// TIA Portal project "N029_Testy Przekladni" (V17)

(* hardware
DEVICE "S7-1200 station_1"  S7-1200 Station
   slot 0: "Rack_0"  S7-1200 Rack  Rack  V1.0
   slot 1: "PLC"  CPU 1212C DC/DC/DC  6ES7 212-1AE40-0XB0  V4.5
DEVICE "HMI"  TP1200 Comfort
   slot 0: "HMI"  TP1200 Comfort  6AV2 124-0MC01-0AX0  17.0.0.0
   slot 1: "HMI_RT_1"  TP1200 Comfort  6AV2 124-0MC01-0AX0  17.0.0.0
   slot 5: "HMI.IE_CP_1"  PROFINET Interface  17.0.0.0
      slot 1: "PROFINET Interface_1"  PROFINET Interface
         slot 1: "Port_1"  Port
         slot 2: "Port_2"  Port
   slot 7: "HMI.MPI/DP_CP_1"  MPI/DP Interface  17.0.0.0
DEVICE "GSD device_1"  GSD.Device.PN
   slot 0: "Rack"  Rack  V1.0
   slot 0: "SK550P-PNT"  SK 550P-PNT
      slot 0: "SK 550P-PNT"  SK 550P-PNT
      slot 1: "PN-IO"  PN-IO
         slot 1: "Port 1 - RJ45 Connector 1"  Port 1 - RJ45 Connector 1
         slot 2: "Port 2 - RJ45 Connector 2"  Port 2 - RJ45 Connector 2
   slot 3: "PPO 4 (4 words)_1"  PPO 4 (4 words)
      slot 0: "PPO 4 (4 words)"  PPO 4 (4 words)
DEVICE "SCALANCE X005"  SCALANCE X-Station
   slot 0: "SCALANCE X rack"  Rail
   slot 0: "Switch_1"  6GK5 005-0BA00-1AB2  V1.0
*)

// ===== PLC "PLC"  CPU 1212C DC/DC/DC =====

VAR_GLOBAL   // PLC tag table "Default tag table"
   "Clock_Byte" AT %MB101 : Byte;
   "Clock_10Hz" AT %M101.0 : Bool;
   "Clock_5Hz" AT %M101.1 : Bool;
   "Clock_2.5Hz" AT %M101.2 : Bool;
   "Clock_2Hz" AT %M101.3 : Bool;
   "Clock_1.25Hz" AT %M101.4 : Bool;
   "Clock_1Hz" AT %M101.5 : Bool;
   "Clock_0.625Hz" AT %M101.6 : Bool;
   "Clock_0.5Hz" AT %M101.7 : Bool;
   "System_Byte" AT %MB100 : Byte;
   "FirstScan" AT %M100.0 : Bool;
   "DiagStatusUpdate" AT %M100.1 : Bool;
   "AlwaysTRUE" AT %M100.2 : Bool;
   "AlwaysFALSE" AT %M100.3 : Bool;
   "HMI_screen_no" AT %MB96 : USInt;
   "RUN_AUTO_mode" AT %M10.0 : Bool;
   "HMI_AUTO_Start_auto" AT %M10.2 : Bool;
   "HMI_Stop_auto" AT %M10.3 : Bool;
   "RUN_MANUAL_mode" AT %M10.1 : Bool;
   "MANUAL_direction" AT %M10.4 : Bool;
   "HMI_MANUAL_Start" AT %M10.5 : Bool;
END_VAR

VAR_GLOBAL   // PLC tag table "IOs_tags"
   "IN_pb_Reset" AT %I0.4 : Bool;
   "IN_pb_Start" AT %I0.0 : Bool;
   "OUT_green_LED" AT %M151.5 : Bool;
   "OUT_yellow_LED" AT %M151.6 : Bool;
   "OUT_red_LED" AT %M151.7 : Bool;
   "IN_pb_Gate_2_open" AT %I0.3 : Bool;
   "OUT_Gate_locks" AT %M151.0 : Bool;
   "OUT_pb_Reset_LED" AT %M151.1 : Bool;
   "OUT_pb_Start_LED" AT %M151.2 : Bool;
   "IN_pb_Stop" AT %I0.1 : Bool;
   "AIN_set_speed" AT %IW64 : Int;
   "IN_safety_lock_gate1" AT %I0.5 : Bool;
   "IN_safety_lock_gate2" AT %I0.6 : Bool;
   "IN_pb_Gate_1_open" AT %I0.2 : Bool;
END_VAR

// folder: Common

TYPE "typeDiagnostics"
TITLE = typeDiagnostics
// Provides a structure for detailed diagnostics
   STRUCT
      status : Word;   // Status of the block or error identification when error occurred
      subfunctionStatus : DWord;   // Status or return value of called FBs, FCs and system blocks
      stateNumber : DInt;   // State in the state machine of the block where the error occurred
   END_STRUCT;
END_TYPE

// folder: (top level)

DATA_BLOCK "Prozess_PPO2/4_DB"   // DB2
{ S7_Optimized_Access := 'TRUE' }
VERSION : 0.1
// stored: InstanceOfName Prozess_PPO2/4
"Prozess_PPO2/4"
BEGIN
END_DATA_BLOCK

DATA_BLOCK "Recipe_db"   // DB3
{ S7_Optimized_Access := 'TRUE' }
VERSION : 0.1
   VAR
      Velocity_array : Array[0..13] of Int;
      Time_array : Array[0..13] of Int;
      Set_speed : Int;
      Manual_speed : Int;
      Cumulated_time_array : Array[0..13] of Int;
   END_VAR
BEGIN
END_DATA_BLOCK

DATA_BLOCK "PLC_ variables"   // DB5
{ S7_Optimized_Access := 'TRUE' }
VERSION : 0.1
   VAR RETAIN
      RESET_state : USInt;
      STANDBY_state : USInt := 1;
      CHECK_LOCKS_state : USInt := 4;
      AUTO_state : USInt := 2;
      MANUAL_State : USInt := 3;
   END_VAR
   VAR
      STATE_machine_step : USInt;
      Measured_speed : Int;
   END_VAR
BEGIN
END_DATA_BLOCK

DATA_BLOCK "Auto_mode_DB"   // DB6
{ S7_Optimized_Access := 'TRUE' }
VERSION : 0.1
// stored: InstanceOfName Auto_mode
"Auto_mode"
BEGIN
END_DATA_BLOCK

// folder: System blocks/Program resources

DATA_BLOCK "IEC_Timer_0_DB"   // DB4
{ S7_Optimized_Access := 'TRUE' }
AUTHOR : Simatic
FAMILY : IEC
NAME : IEC_TMR
VERSION : 1.0
// stored: InstanceOfName IEC_TIMER
"IEC_TIMER"
BEGIN
END_DATA_BLOCK

DATA_BLOCK "time_from_Start_timer_DB"   // DB7
{ S7_Optimized_Access := 'TRUE' }
AUTHOR : Simatic
FAMILY : IEC
NAME : UDCNTR
VERSION : 1.2
// stored: InstanceOfName IEC_UDCOUNTER
"IEC_UDCOUNTER"
BEGIN
END_DATA_BLOCK

DATA_BLOCK "IEC_Counter_0_DB"   // DB8
{ S7_Optimized_Access := 'TRUE' }
AUTHOR : Simatic
FAMILY : IEC
NAME : CNTR
VERSION : 1.0
// stored: InstanceOfName IEC_COUNTER
"IEC_COUNTER"
BEGIN
END_DATA_BLOCK

DATA_BLOCK "IEC_Timer_0_DB_1"   // DB9
{ S7_Optimized_Access := 'TRUE' }
AUTHOR : Simatic
FAMILY : IEC
NAME : IEC_TMR
VERSION : 1.0
// stored: InstanceOfName IEC_TIMER
"IEC_TIMER"
BEGIN
END_DATA_BLOCK

// folder: (top level)

FUNCTION_BLOCK "Auto_mode"   // FB1, LAD
{ S7_Optimized_Access := 'TRUE' }
VERSION : 0.1
   VAR_OUTPUT
      Set_speed : Int;
   END_VAR
   VAR
      "60sec_marker" : Bool;
      STOPPED : USInt := 3;
      BRAKE : USInt := 2;
      RUN : USInt := 1;
      PREPARE_VAL : USInt;
      Time_from_start : UDInt;
      Time_for_next_step : UDInt;
      State : USInt;
   END_VAR
   VAR_TEMP
      "60sec" : Bool;
      timer_reset_marker : Bool;
      Time_curr_step : Int;
      Time_next_step : Int;
      i : Int;
      Curr_set_velocity : Int;
      Next_set_velocity : Int;
      j : Int;
      dVelocity : Int;
      Time_Step : Real;
      dTime : Real;
   END_VAR
BEGIN

REGION Network 1
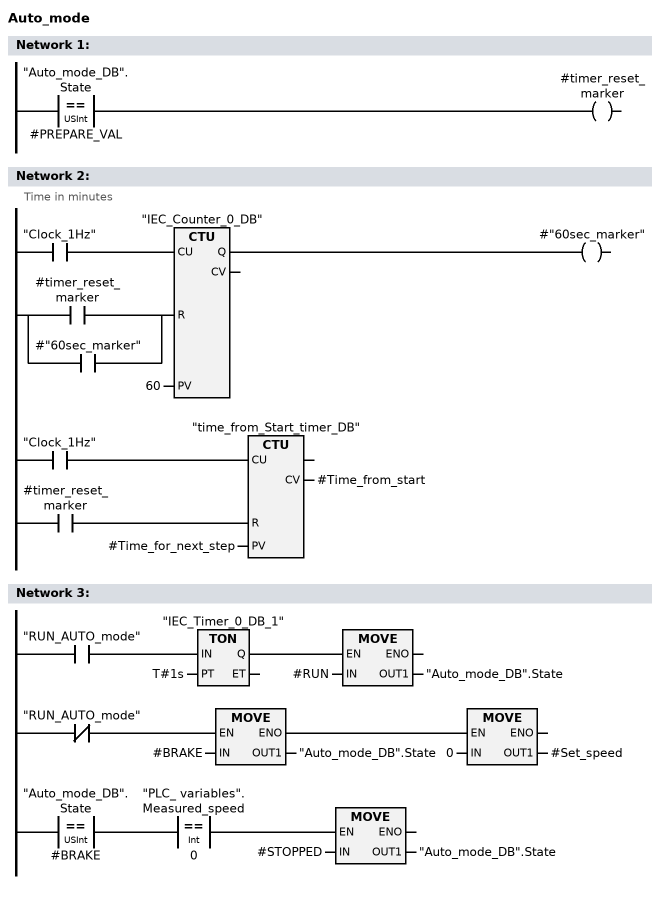
   RUNG wire#powerrail
      { S7_Templates := "SrcType := USInt" } EQ_Contact(in1 := "Auto_mode_DB".State, in2 := #PREPARE_VAL)
      Coil( #timer_reset_marker )
   END_RUNG
   // the same network as SCL:
   #timer_reset_marker := "Auto_mode_DB".State = #PREPARE_VAL;
END_REGION

REGION Network 2
   // Time in minutes
   "IEC_Counter_0_DB".CTU(CU := "Clock_1Hz", R := #timer_reset_marker OR #"60sec_marker", PV := 60);
   #"60sec_marker" := "IEC_Counter_0_DB".Q;
   "time_from_Start_timer_DB".CTU(CU := "Clock_1Hz",
                           R := #timer_reset_marker,
                           PV := #Time_for_next_step,
                           CV => #Time_from_start);
END_REGION

REGION Network 3
   "IEC_Timer_0_DB_1".TON(IN := "RUN_AUTO_mode", PT := T#1s);
   IF "IEC_Timer_0_DB_1".Q THEN "Auto_mode_DB".State := #RUN; END_IF;
   IF NOT "RUN_AUTO_mode" THEN
       "Auto_mode_DB".State := #BRAKE;
       #Set_speed := 0;
   END_IF;
   IF ("Auto_mode_DB".State = #BRAKE) AND ("PLC_ variables".Measured_speed = 0) THEN
       "Auto_mode_DB".State := #STOPPED;
   END_IF;
END_REGION

REGION Network 4 (SCL)
   IF (#State = #RUN OR #State = #PREPARE_VAL) THEN

       "Recipe_db".Cumulated_time_array[0] := 0;

       FOR #i := 0 TO 12 BY 1 DO
           "Recipe_db".Cumulated_time_array[#i + 1] := "Recipe_db".Cumulated_time_array[#i] + "Recipe_db".Time_array[#i + 1];
       END_FOR;

       FOR #j := 0 TO 12 BY 1 DO
           IF (#Time_from_start < ("Recipe_db".Cumulated_time_array[#j + 1] * 60)) THEN
               #Time_curr_step := "Recipe_db".Cumulated_time_array[#j] * 60;
               #Time_next_step := "Recipe_db".Cumulated_time_array[#j + 1] * 60;
               #Curr_set_velocity := "Recipe_db".Velocity_array[#j];
               #Next_set_velocity := "Recipe_db".Velocity_array[#j + 1];
               EXIT;
           ELSIF  (#Time_from_start > ("Recipe_db".Cumulated_time_array[#j + 1] * 60) AND #i=12) THEN
               #State:=#BRAKE;
           END_IF;
       END_FOR;

       #dTime := UDINT_TO_REAL(#Time_from_start - INT_TO_UDINT(#Time_curr_step));
       #Time_Step := (#Time_next_step - #Time_curr_step);
       #dVelocity := (#Next_set_velocity - #Curr_set_velocity);
       #Set_speed := #Curr_set_velocity + REAL_TO_INT(#dVelocity * (#dTime / #Time_Step));
   END_IF;
END_REGION
END_FUNCTION_BLOCK

FUNCTION_BLOCK "Prozess_PPO2/4"   // FB2, SCL
TITLE = PPO2/4
{ S7_Optimized_Access := 'TRUE' }
VERSION : 0.1
   VAR_INPUT
      HW_Identifier : Hw_Io;   // unique system constant created automatically by the system
      FI_Systembus : Int := 1;   // for frequency inverters in a system bus (1..8)
      Enable : Bool;   // 1 = enable drive
      Disable_Voltage : Bool;   // 1 = disable voltage
      Quick_Stop : Bool;   // 1 = quick stop
      Fault_ACK : Bool;   // 0 -> 1 fault acknowledgement
      Function_CTW_8 : Bool;   // bus controlword bit 8
      Function_CTW_9 : Bool;   // bus controlword bit 9
      Direction : Bool;   // 0 = cw / 1 = ccw
      Parameter_Set : Int;   // set of parameter (1..4)
      Setpoint_1 : Int;   // value setpoint 1
      Setpoint_2 : Int;   // value setpoint 2
      Setpoint_3 : Int;   // value setpoint 3
      Setpoint_32_Bit : Bool;   // 0 = setpoint 2 (16 bit) + setpoint 3 (16 bit) / 1 = setpoint 2 + 3 (32 bit)
      Setpoint_2_3 : DInt;   // value setpoint 2 + 3 (32 bit)
   END_VAR
   VAR_OUTPUT
      Not_Ready_to_Switch_On : Bool;   // inverter in not ready to switch-on state
      Switch_On_Inhibit : Bool;   // inverter in switch-on inhibit state
      Ready_to_Switch_On : Bool;   // inverter in ready to switch-on state
      Operation_Enabled : Bool;   // inverter in operation enabled state
      Fault : Bool;   // inverter in fault state
      Fault_Active : Bool;   // inverter in fault active state
      Quick_Stop_Active : Bool;   // inverter in quick stop active state
      Warning : Bool;   // warning identified
      Function_STW_10 : Bool;   // bus statusword bit 10
      Function_STW_13 : Bool;   // bus statusword bit 13
      Actual_Parameter_Set : Int;   // actual set of parameter 1..4
      Statusword : Word;   // statusword from inverter
      Actual_Value_1 : Int;   // actual value 1
      Actual_Value_2 : Int;   // actual value 2
      Actual_Value_3 : Int;   // actual value 3
      Actual_Value_2_3 : DInt;   // actual value 2 + 3 (32 bit)
   END_VAR
   VAR
      Controlword_Static : Word;   // controlword (to inverter)
      Control AT Controlword_Static : Struct   // definition controlword bits
         Start_Function_CTW_8 : Bool;   // set controlword bit 8
         Start_Function_CTW_9 : Bool;   // set controlword bit 9
         PZD_Valid : Bool;   // 0 = the transmitted data are invalid; 1 = the bus master transfers valid process data
         Rotatation_CW : Bool;   // 1 = switch on clockwise rotation
         Rotatation_CCW : Bool;   // 1 = switch on counter clockwise rotation
         Reserved : Bool;   // reserved
         Parameter_Set_Bit_0 : Bool;   // bit 0 of parameter set selection
         Parameter_Set_Bit_1 : Bool;   // bit 1 of parameter set selection
         Ready_for_Operation : Bool;   // 0 = reverse with break ramp, with voltage enabled at f=0Hz; 1 = set the frequency inverter to standby
         Disable_Voltage : Bool;   // 0 = switch off the output voltage; 1 = cancel "disable voltage"
         Quick_Stop : Bool;   // 0 = quick stop with programmed quick stop time; 1 = cancel "quick stop"
         Enable_Operation : Bool;   // 0 = block voltage; 1 = enable output voltage acceleration to acual setpoint
         Enable_Pulses : Bool;   // 0 = disable frequency inverter pulses; 1 = enable frequency inverter pulses
         Enable_Ramp : Bool;   // 0 = freeze actual frequency; 1 = enable frequency ramp
         Enable_Setpoint : Bool;   // 0 = set the setpoint to zero; 1 = use actual setpoint
         Acknowledge_the_Error : Bool;   // with the switch from 0 to 1, inactive errors are acknowledged
      END_STRUCT;
      GeoAddr : GEOADDR;   // geoaddr of the slot
      Get_GeoAddr : GEOADDR;   // geoaddr of the ~head module
      Statusword_Static : Word;   // statusword (from inverter)
      Status AT Statusword_Static : Struct   // definition statusword bits
         Setpoint_Reached : Bool;   // 0 = actual value does not correspond to the setpoint; 1 = actual value matches the setpoint
         Bus_Control : Bool;   // 0 = control on local device active; 1 = the master has been requested to take over control
         Function_STW_10 : Bool;   // function statusword bit 10 is active
         Rotatation_CW : Bool;   // 1 = the rotating field is clockwise
         Rotatation_CCW : Bool;   // 1 = the rotating field is counter-clockwise
         Function_STW_13 : Bool;   // function statusword bit 13 is active
         Parameter_Set_Bit_0 : Bool;   // bit 0 of the actual parameter set
         Parameter_Set_Bit_1 : Bool;   // bit 1 of the actual parameter set
         Ready_to_Switch_On : Bool;   // 1 = initialisation completed, charging relay switched on, output voltage disabled
         Ready : Bool;   // 0 = no switch-on command present or there is a fault; 1 = there is a switch-on command and there is no fault
         Operation_Enabled : Bool;   // 1 = the output voltage is enabled
         Fault : Bool;   // 0 = no fault 1 = the frequency inverter is in fault
         Voltage_Enabled : Bool;   // 0 = "disable voltage" command present
         Quick_Stop : Bool;   // 0 = "quick stop" command present
         Switch_On_Inhibit : Bool;   // 1 = with the command "shut down" the frequency inverter goes into state "ready to switch-on"
         Warning : Bool;   // 0 = no warning; 1 = active warning; drive operation continues, no acknowledgement necessary
      END_STRUCT;
   END_VAR
   VAR_TEMP
      Input_Address : DInt;   // input address of bus module
      Iw_Fi : UDInt;   // input start address from hardware configurator
      Iw_Fi_Length : UDInt;   // number of input bytes
      Laddr : Hw_Any;   // slot hw address
      Output_Address : DInt;   // output address of bus module
      Qw_Fi : UDInt;   // output start address from hardware configurator
      Qw_Fi_Length : UDInt;   // number of output bytes
      Ret_Geo2Log : Int;   // gro2log error information
      Ret_Log2Geo : Int;   // log2geo error information
      Ret_Rd_Addr : Int;   // rd_addr error information
   END_VAR
   VAR CONSTANT
      NOT_READY_TO_SWITCH_ON_MASK : Word := 2#1001111;   // status word mask for not ready to switch on
      NOT_READY_TO_SWITCH_ON_STATE : Word := 2#0000000;   // decoded fi status not ready to switch on
      SWITCH_ON_INHIBIT_MASK : Word := 2#1001111;   // status word mask for switch on inhibit
      SWITCH_ON_INHIBIT_STATE : Word := 2#1000000;   // decoded fi status switch on inhibit
      READY_TO_SWITCH_ON_MASK : Word := 2#1111111;   // status word mask for ready to swtich on
      READY_TO_SWITCH_ON_STATE : Word := 2#0110001;   // decoded fi status ready to swtich on
      SWITCHED_ON_MASK : Word := 2#1111111;   // status word mask for switched on
      SWITCHED_ON_STATE : Word := 2#0110011;   // decoded fi status switched on
      OPERATION_ENABLED_MASK : Word := 2#1111111;   // status word mask for operation enabled
      OPERATION_ENABLED_STATE : Word := 2#0110111;   // decoded fi status operation enabled
      FAULT_MASK : Word := 2#1001111;   // status word mask for fault
      FAULT_STATE : Word := 2#0001000;   // decoded fi status fault
      FAULT_ACTIVE_MASK : Word := 2#1001111;   // status word mask for fault activ
      FAULT_ACTIVE_STATE : Word := 2#0001111;   // decoded fi status fault activ
      PPO2_LENGTH : Word := 16;   // length of a ppo2 frame
      PPO2_4_LENGTH_TU3_PBR : Word := 12;   // length of a ppo2 and ppo4 pzd frame for a sk tu3-pbr
      PPO4_LENGTH : Word := 8;   // length of a ppo4 frame
      PROFIBUS : UInt := 2;   // profibus dp geoaddr area
      PROFINET : UInt := 1;   // profinet io geoaddr area
      QUICK_STOP_ACTIVE_MASK : Word := 2#1111111;   // status word mask for quick stop activ
      QUICK_STOP_ACTIVE_STATE : Word := 2#0010111;   // decoded fi status quick stop activ
      SLOT_OFFSET_PBR : UInt := 1;   // profibus dp slot offset of bus module
      SLOT_OFFSET_PNT : UInt := 2;   // profinet io slot offset of bus module
   END_VAR
   // GeoAddr.HWTYPE := 4;
BEGIN
   // get area, io station and station from ~head module (hw address)
   #Ret_Log2Geo := LOG2GEO(LADDR := #HW_Identifier, GEOADDR := #Get_GeoAddr);
   #GeoAddr.AREA := #Get_GeoAddr.AREA;
   #GeoAddr.IOSYSTEM := #Get_GeoAddr.IOSYSTEM;
   #GeoAddr.STATION := #Get_GeoAddr.STATION;

   IF #Get_GeoAddr.AREA = #PROFINET THEN     // for profinet io
       #GeoAddr.SLOT := INT_TO_UINT(#FI_Systembus) + #SLOT_OFFSET_PNT;
   ELSIF #Get_GeoAddr.AREA = #PROFIBUS THEN  // for profibus dp
       #GeoAddr.SLOT := INT_TO_UINT(#FI_Systembus) + #SLOT_OFFSET_PBR;
   ELSE  // wrong area
       #Actual_Value_1 := 0;
       #Actual_Value_2 := 0;
       #Actual_Value_3 := 0;
       #Actual_Value_2_3 := 0;
       #Not_Ready_to_Switch_On := FALSE;
       #Switch_On_Inhibit := FALSE;
       #Ready_to_Switch_On := FALSE;
       #Operation_Enabled := FALSE;
       #Fault_Active := FALSE;
       #Fault := FALSE;
       #Quick_Stop_Active := FALSE;
       #Warning := FALSE;
       #Function_STW_10 := FALSE;
       #Function_STW_13 := FALSE;
       #Statusword := 0;
       #Actual_Parameter_Set := 0;
       RETURN;
   END_IF;

   // get slot hw address (systembus fi)
   #Ret_Geo2Log := GEO2LOG(GEOADDR := #GeoAddr, LADDR => #Laddr);
   // based on slot hw address get io addresses
   #Ret_Rd_Addr := RD_ADDR(LADDR := #Laddr, PIADDR => #Iw_Fi, PICount => #Iw_Fi_Length,
                           PQADDR => #Qw_Fi, PQCount => #Qw_Fi_Length);

   IF #Iw_Fi_Length = #PPO4_LENGTH THEN    // if PPO4 -> no PKW channel
       #Input_Address  := UDINT_TO_DINT(#Iw_Fi);
       #Output_Address := UDINT_TO_DINT(#Qw_Fi);
   ELSIF #Iw_Fi_Length = #PPO2_4_LENGTH_TU3_PBR AND
         #Get_GeoAddr.AREA = #PROFIBUS THEN // special case SK xU3-PBR: PPO2/4 -> 6 words/no PKW channel
       #Input_Address := UDINT_TO_DINT(#Iw_Fi);
       #Output_Address := UDINT_TO_DINT(#Qw_Fi);
   ELSIF #Iw_Fi_Length = #PPO2_LENGTH THEN  // else if PPO2 -> with PKW channel
       #Input_Address  := UDINT_TO_DINT(#Iw_Fi) + 8;
       #Output_Address := UDINT_TO_DINT(#Qw_Fi) + 8;
   ELSE // wrong PPO Type
       #Actual_Value_1 := 0;
       #Actual_Value_2 := 0;
       #Actual_Value_3 := 0;
       #Actual_Value_2_3 := 0;
       #Not_Ready_to_Switch_On := FALSE;
       #Switch_On_Inhibit := FALSE;
       #Ready_to_Switch_On := FALSE;
       #Operation_Enabled := FALSE;
       #Fault_Active := FALSE;
       #Fault := FALSE;
       #Quick_Stop_Active := FALSE;
       #Warning := FALSE;
       #Function_STW_10 := FALSE;
       #Function_STW_13 := FALSE;
       #Statusword := 0;
       #Actual_Parameter_Set := 0;
       RETURN;
   END_IF;

   // prepare controlword to inverter********************
   #Control.Ready_for_Operation    := #Enable;
   #Control.Disable_Voltage        := NOT #Disable_Voltage;
   #Control.Quick_Stop             := NOT #Quick_Stop;
   #Control.Enable_Operation       := TRUE;
   #Control.Enable_Pulses          := TRUE;
   #Control.Enable_Ramp            := TRUE;
   #Control.Enable_Setpoint        := TRUE;
   #Control.Acknowledge_the_Error  := #Fault_ACK;
   #Control.Start_Function_CTW_8   := #Function_CTW_8;
   #Control.Start_Function_CTW_9   := #Function_CTW_9;
   #Control.PZD_Valid              := TRUE;
   #Control.Rotatation_CCW         := #Direction;

   CASE #Parameter_Set OF
       1:  // statement section parameter set 1
           #Control.Parameter_Set_Bit_0 := FALSE;
           #Control.Parameter_Set_Bit_1 := FALSE;
       2:  // statement section parameter set 2
           #Control.Parameter_Set_Bit_0 := TRUE;
           #Control.Parameter_Set_Bit_1 := FALSE;
       3:  // statement section parameter set 3
           #Control.Parameter_Set_Bit_0 := FALSE;
           #Control.Parameter_Set_Bit_1 := TRUE;
       4:  // statement section parameter set 4
           #Control.Parameter_Set_Bit_0 := TRUE;
           #Control.Parameter_Set_Bit_1 := TRUE;
       ELSE  // default statement section parameter set 1
           #Control.Parameter_Set_Bit_0 := FALSE;
           #Control.Parameter_Set_Bit_1 := FALSE;
   END_CASE;

   // write controlword**********************************
   POKE(area := 16#82,
        dbNumber := 0,
        byteOffset := #Output_Address,
        value := #Controlword_Static);
   // write setpoints************************************
   POKE(area := 16#82,
        dbNumber := 0,
        byteOffset := #Output_Address + 2,
        value := INT_TO_WORD(#Setpoint_1));
   IF #Setpoint_32_Bit THEN
       POKE(area := 16#82,
            dbNumber := 0,
            byteOffset := #Output_Address + 4,
            value := DINT_TO_DWORD(#Setpoint_2_3));
   ELSE
       POKE(area := 16#82,
            dbNumber := 0,
            byteOffset := #Output_Address + 4,
            value := INT_TO_WORD(#Setpoint_2));
       POKE(area := 16#82,
            dbNumber := 0,
            byteOffset := #Output_Address + 6,
            value := INT_TO_WORD(#Setpoint_3));
   END_IF;

   // read statusword************************************
   #Statusword_Static := PEEK_WORD(area := 16#81, dbNumber := 0, byteOffset := #Input_Address);
   // read actual values*********************************
   #Actual_Value_1   := WORD_TO_INT(PEEK_WORD(area := 16#81, dbNumber := 0, byteOffset := #Input_Address + 2));
   #Actual_Value_2   := WORD_TO_INT(PEEK_WORD(area := 16#81, dbNumber := 0, byteOffset := #Input_Address + 4));
   #Actual_Value_3   := WORD_TO_INT(PEEK_WORD(area := 16#81, dbNumber := 0, byteOffset := #Input_Address + 6));
   #Actual_Value_2_3 := DWORD_TO_DINT(PEEK_DWORD(area := 16#81, dbNumber := 0, byteOffset := #Input_Address + 4));

   // decode statusword and set outputs******************
   #Not_Ready_to_Switch_On := (#Statusword_Static AND #NOT_READY_TO_SWITCH_ON_MASK) = #NOT_READY_TO_SWITCH_ON_STATE;
   #Switch_On_Inhibit      := (#Statusword_Static AND #SWITCH_ON_INHIBIT_MASK) = #SWITCH_ON_INHIBIT_STATE;
   #Ready_to_Switch_On     := (#Statusword_Static AND #READY_TO_SWITCH_ON_MASK) = #READY_TO_SWITCH_ON_STATE;
   #Operation_Enabled      := (#Statusword_Static AND #OPERATION_ENABLED_MASK) = #OPERATION_ENABLED_STATE;
   #Fault_Active           := (#Statusword_Static AND #FAULT_ACTIVE_MASK) = #FAULT_ACTIVE_STATE;
   #Fault                  := (#Statusword_Static AND #FAULT_MASK) = #FAULT_STATE;
   #Quick_Stop_Active      := (#Statusword_Static AND #QUICK_STOP_ACTIVE_MASK) = #QUICK_STOP_ACTIVE_STATE;
   #Warning                := #Status.Warning;
   #Function_STW_10        := #Status.Function_STW_10;
   #Function_STW_13        := #Status.Function_STW_13;
   #Statusword             := #Statusword_Static;
   #Actual_Parameter_Set   := WORD_TO_INT(SHR(IN := #Statusword_Static, N := 14)) + 1;
END_FUNCTION_BLOCK

FUNCTION "Manual_mode" : Void   // FC1, LAD
{ S7_Optimized_Access := 'TRUE' }
VERSION : 0.1
   VAR_OUTPUT
      Set_speed : Int;
   END_VAR
   VAR_TEMP
      calculated_speed : Real;
   END_VAR
   VAR CONSTANT
      MULTIPLY : Real := 0.2;
   END_VAR
BEGIN

REGION Network 1 (SCL)
   #calculated_speed := INT_TO_REAL("AIN_set_speed") * #MULTIPLY;
   #Set_speed := REAL_TO_INT(LIMIT_REAL(IN:=#calculated_speed,MN:= 0.0,MX:= 6000.0));
END_REGION
END_FUNCTION

ORGANIZATION_BLOCK "Main"   // OB1, LAD, ProgramCycle
TITLE = "Main Program Sweep (Cycle)"
{ S7_Optimized_Access := 'TRUE' }
VERSION : 0.1
   VAR_INPUT
      Initial_Call : Bool;   // Initial call of this OB
      Remanence : Bool;   // =True, if remanent data are available
   END_VAR
   VAR_TEMP   // added for the SCL form of the ladder/FBD networks
      _w1 : Bool;
   END_VAR
BEGIN

REGION Network 1: initial state
   // State machine
   // 1- reset state
   // 2- standby
   // 3- manual mode
   // 4- auto mode
   // 5- error
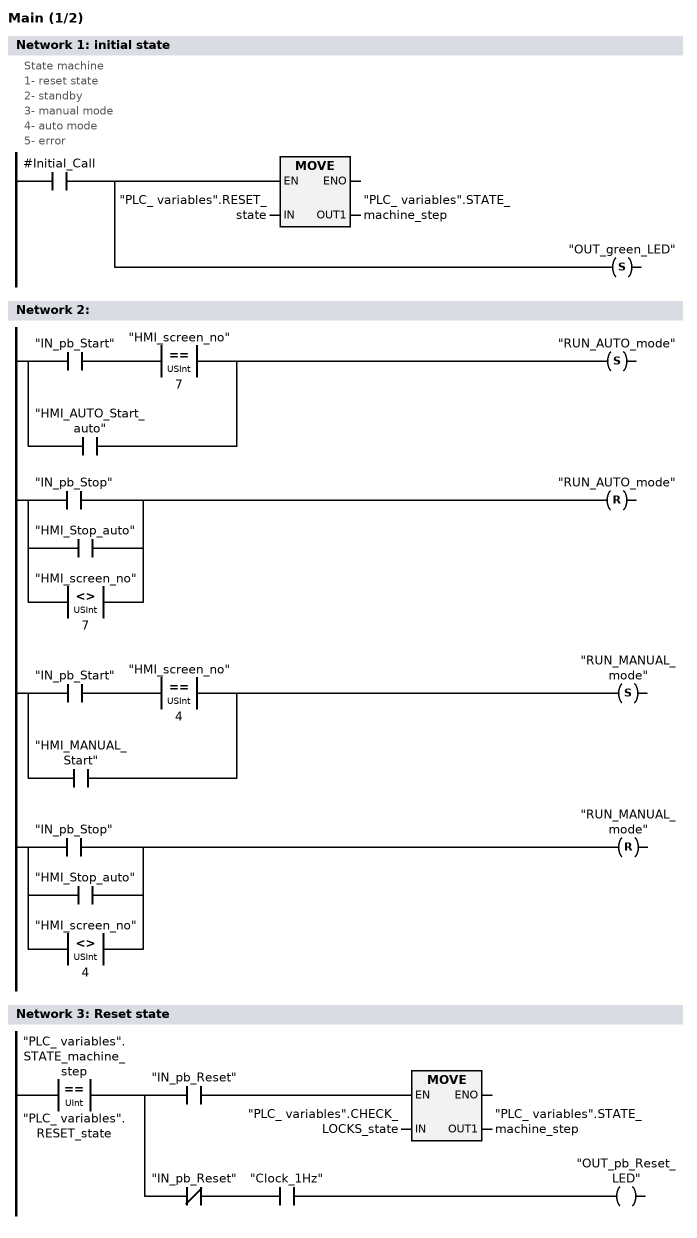
   RUNG wire#powerrail
      Contact( #Initial_Call )
      wire#w1
      Move(in := "PLC_ variables".RESET_state, out1 => "PLC_ variables".STATE_machine_step)
   END_RUNG
   RUNG wire#w1
      S_Coil( "OUT_green_LED" )
   END_RUNG
   // the same network as SCL:
   IF #Initial_Call THEN
       "PLC_ variables".STATE_machine_step := "PLC_ variables".RESET_state;
       "OUT_green_LED" := TRUE;
   END_IF;
END_REGION

REGION Network 2
   RUNG wire#powerrail
      Contact( "IN_pb_Start" )
      { S7_Templates := "SrcType := USInt" } EQ_Contact(in1 := "HMI_screen_no", in2 := 7)
      wire#w1
      S_Coil( "RUN_AUTO_mode" )
   END_RUNG
   RUNG wire#powerrail
      Contact( "HMI_AUTO_Start_auto" )
   END_RUNG wire#w1
   RUNG wire#powerrail
      Contact( "IN_pb_Stop" )
      wire#w2
      R_Coil( "RUN_AUTO_mode" )
   END_RUNG
   RUNG wire#powerrail
      Contact( "HMI_Stop_auto" )
   END_RUNG wire#w2
   RUNG wire#powerrail
      { S7_Templates := "SrcType := USInt" } NE_Contact(in1 := "HMI_screen_no", in2 := 7)
   END_RUNG wire#w2
   RUNG wire#powerrail
      Contact( "IN_pb_Start" )
      { S7_Templates := "SrcType := USInt" } EQ_Contact(in1 := "HMI_screen_no", in2 := 4)
      wire#w3
      S_Coil( "RUN_MANUAL_mode" )
   END_RUNG
   RUNG wire#powerrail
      Contact( "HMI_MANUAL_Start" )
   END_RUNG wire#w3
   RUNG wire#powerrail
      Contact( "IN_pb_Stop" )
      wire#w4
      R_Coil( "RUN_MANUAL_mode" )
   END_RUNG
   RUNG wire#powerrail
      Contact( "HMI_Stop_auto" )
   END_RUNG wire#w4
   RUNG wire#powerrail
      { S7_Templates := "SrcType := USInt" } NE_Contact(in1 := "HMI_screen_no", in2 := 4)
   END_RUNG wire#w4
   // the same network as SCL:
   IF ("IN_pb_Start" AND ("HMI_screen_no" = 7)) OR "HMI_AUTO_Start_auto" THEN
       "RUN_AUTO_mode" := TRUE;
   END_IF;
   IF "IN_pb_Stop" OR "HMI_Stop_auto" OR ("HMI_screen_no" <> 7) THEN "RUN_AUTO_mode" := FALSE; END_IF;
   IF ("IN_pb_Start" AND ("HMI_screen_no" = 4)) OR "HMI_MANUAL_Start" THEN "RUN_MANUAL_mode" := TRUE; END_IF;
   IF "IN_pb_Stop" OR "HMI_Stop_auto" OR ("HMI_screen_no" <> 4) THEN "RUN_MANUAL_mode" := FALSE; END_IF;
END_REGION

REGION Network 3: Reset state
   RUNG wire#powerrail
      { S7_Templates := "SrcType := UInt" } EQ_Contact(in1 := "PLC_ variables".STATE_machine_step, in2 := "PLC_ variables".RESET_state)
      wire#w1
      Contact( "IN_pb_Reset" )
      Move(in := "PLC_ variables".CHECK_LOCKS_state, out1 => "PLC_ variables".STATE_machine_step)
   END_RUNG
   RUNG wire#w1
      I_Contact( "IN_pb_Reset" )
      Contact( "Clock_1Hz" )
      Coil( "OUT_pb_Reset_LED" )
   END_RUNG
   // the same network as SCL:
   #_w1 := "PLC_ variables".STATE_machine_step = "PLC_ variables".RESET_state;
   IF #_w1 AND "IN_pb_Reset" THEN
       "PLC_ variables".STATE_machine_step := "PLC_ variables".CHECK_LOCKS_state;
   END_IF;
   "OUT_pb_Reset_LED" := #_w1 AND NOT "IN_pb_Reset" AND "Clock_1Hz";
END_REGION

REGION Network 5: Standby state
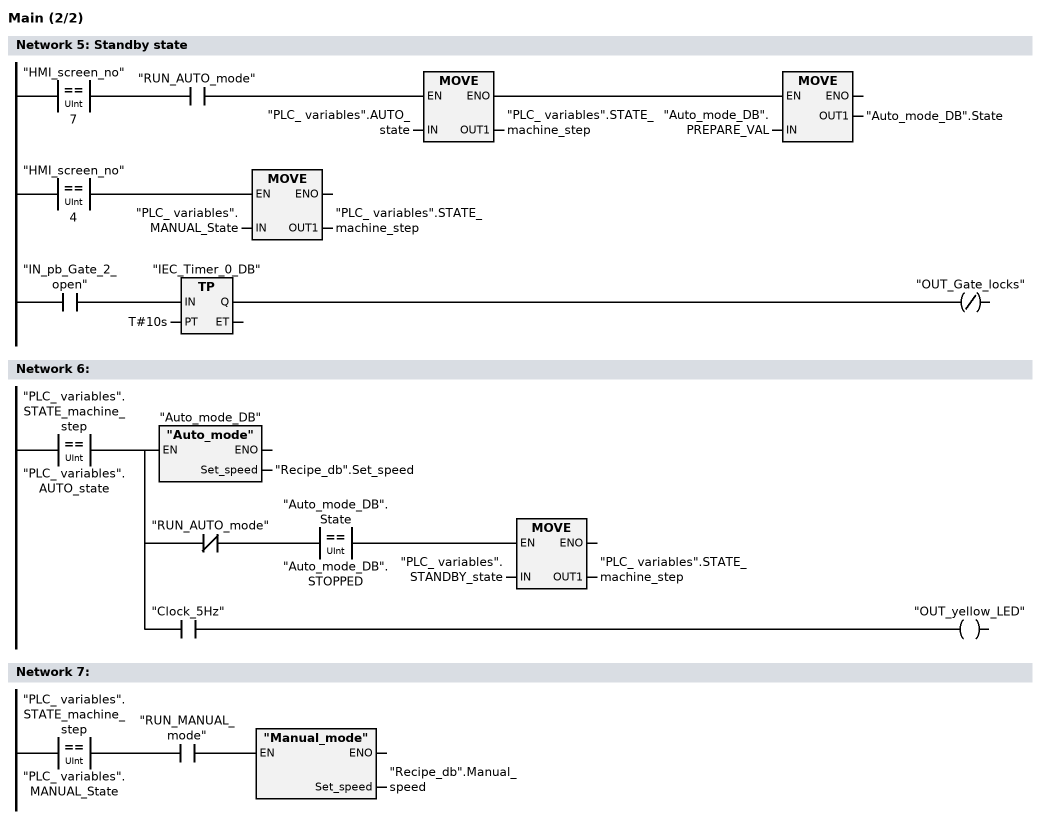
   IF ("HMI_screen_no" = 7) AND "RUN_AUTO_mode" THEN
       "PLC_ variables".STATE_machine_step := "PLC_ variables".AUTO_state;
       "Auto_mode_DB".State := "Auto_mode_DB".PREPARE_VAL;
   END_IF;
   IF "HMI_screen_no" = 4 THEN "PLC_ variables".STATE_machine_step := "PLC_ variables".MANUAL_State; END_IF;
   "IEC_Timer_0_DB".TP(IN := "IN_pb_Gate_2_open", PT := T#10s);
   "OUT_Gate_locks" := NOT "IEC_Timer_0_DB".Q;
END_REGION

REGION Network 6
   RUNG wire#powerrail
      { S7_Templates := "SrcType := UInt" } EQ_Contact(in1 := "PLC_ variables".STATE_machine_step, in2 := "PLC_ variables".AUTO_state)
      wire#w1
      "Auto_mode_DB"(Set_speed => "Recipe_db".Set_speed)
   END_RUNG
   RUNG wire#w1
      I_Contact( "RUN_AUTO_mode" )
      { S7_Templates := "SrcType := UInt" } EQ_Contact(in1 := "Auto_mode_DB".State, in2 := "Auto_mode_DB".STOPPED)
      Move(in := "PLC_ variables".STANDBY_state, out1 => "PLC_ variables".STATE_machine_step)
   END_RUNG
   RUNG wire#w1
      Contact( "Clock_5Hz" )
      Coil( "OUT_yellow_LED" )
   END_RUNG
   // the same network as SCL:
   #_w1 := "PLC_ variables".STATE_machine_step = "PLC_ variables".AUTO_state;
   IF #_w1 THEN
       "Auto_mode_DB"(Set_speed => "Recipe_db".Set_speed);   // "Auto_mode"
   END_IF;
   IF #_w1 AND NOT "RUN_AUTO_mode" AND ("Auto_mode_DB".State = "Auto_mode_DB".STOPPED) THEN
       "PLC_ variables".STATE_machine_step := "PLC_ variables".STANDBY_state;
   END_IF;
   "OUT_yellow_LED" := #_w1 AND "Clock_5Hz";
END_REGION

REGION Network 7
   RUNG wire#powerrail
      { S7_Templates := "SrcType := UInt" } EQ_Contact(in1 := "PLC_ variables".STATE_machine_step, in2 := "PLC_ variables".MANUAL_State)
      Contact( "RUN_MANUAL_mode" )
      "Manual_mode"(Set_speed => "Recipe_db".Manual_speed)
   END_RUNG
   // the same network as SCL:
   IF ("PLC_ variables".STATE_machine_step = "PLC_ variables".MANUAL_State) AND "RUN_MANUAL_mode" THEN
       "Manual_mode"(Set_speed => "Recipe_db".Manual_speed);
   END_IF;
END_REGION
END_ORGANIZATION_BLOCK

// ===== library types =====

// folder: LFTP

TYPE "LFTP_typeFtpParam"
TITLE = LFTP_typeFtpParam / LFTP_typeUserParam
VERSION : 0.1
// Data type for user parameters of the LFTP FB / Data type for user parameters of the LFTP_Client FB
   STRUCT
      ftpActiveMode : Bool;   // False: FTP mode is set to passive; True: FTP mode is set to active
      portActiveMode : UInt := 2001;   // Must be set >2000; Port for FTP-active mode data connection / Must be set >2000; Local Port for FTP active mode
      ftpCmd : Int;   // 2 STORE, 3 RETRIEVE, 4 DELETE, 6 APPEND
      filename : String;   // FTP Filename
   END_STRUCT;
END_TYPE

TYPE "LFTP_typeConnParam"
TITLE = LFTP_typeConnParam
// Datatype for the Parameters needed for connection to FTP-Server / Data type for connection parameters needed to establish a connection to the FTP server
   STRUCT
      hwID : HW_ANY;   // HW-identifier of IE-interface submodule
      serverAddress : String;   // Remote-Adress of FTP-Server / IP address or host name of FTP server
      username : String := '';   // Username of the FTP-Client / User name of the FTP client
      password : String := '';   // Password of the FTP-Client / Password of the FTP client
   END_STRUCT;
END_TYPE

FUNCTION_BLOCK "LFTP_Client"   // FB2, SCL
TITLE = LFTP_Client
{ S7_Optimized_Access := 'TRUE' }
AUTHOR : Siemens Industry Online Support
FAMILY : LFTP
VERSION : 6.0
// Implements an FTP client
   VAR_INPUT
      enable : Bool := FALSE;   // Enable client and connect to FTP server
      execute : Bool := FALSE;   // Execute FTP command
      timeOut : Time := T#5s;   // Time for watchdog
   END_VAR
   VAR_OUTPUT
      valid : Bool := FALSE;   // TRUE: Valid set of output values available at the FB
      done : Bool := FALSE;   // TRUE: Last command was successful
      busy : Bool := FALSE;   // TRUE: FB is not finished and new output values can be expected
      error : Bool := FALSE;   // TRUE: An error occurred during the execution of the FB
      status : Word := 16#7000;   // 16#0000 - 16#7FFF: Status of the FB, 16#8000 - 16#FFFF: Error identification
      diagnostics : "typeDiagnostics";   // Diagnostics information of FB
   END_VAR
   VAR_IN_OUT
      connParam : "LFTP_typeConnParam";   // Connection parameters
      ftpParam : "LFTP_typeFtpParam";   // FTP parameters
      dataLen : UDInt;   // Length of data to be sent or received
      data : Array[*] of Byte;   // Data to be sent or received
   END_VAR
   VAR
      statEnableOld : Bool;   // Last cycle's value of 'enable' input for edge detection
      statExecuteOld : Bool;   // Last cycle's value of 'execute' input for edge detection
      statValid : Bool;   // Static value for output 'valid'
      statDone : Bool;   // Static value for output 'done'
      statBusy : Bool;   // Static value for output 'busy'
      statError : Bool;   // Static value for output 'error'
      statErrorUserCleared : Bool;   // Error occurred that can only be solved by user; rising edge at enable input necessary
      statErrorAutoCleared : Bool;   // Error occurred that can be acknowledged by FB
      statStatus : Word := 16#7000;   // Static value for output 'status'
      statSubfunctionStatus : DWord;   // Status or return value of called FBs, FCs and system blocks
      statFBErrorState : DInt;   // State in the state machine of the block where the error occurred
      statFBState : UInt := 0;   // State in the state machine of the FB
      statDisablingCompleted : Bool;   // TRUE: Disabling has been completed
      statEmptyDiagnostics : "typeDiagnostics";   // Empty diagnostics information (for initialization purposes only)
      statConnParam : Struct   // Connection parameters
         isQDN : Bool;   // Is set to TRUE when connParam.url recognised as QDN
         paramControlQDN : TCON_QDN;   // Connection parameters in form of QDN
         paramControlIP : TCON_IP_v4;   // Connection parameters in form of IP address
         paramDataQDN : TCON_QDN;   // Connection parameters of data connection in form of QDN
         paramDataIP : TCON_IP_v4;   // Connection parameters of data connection in form of IP address
      END_STRUCT;
      statFtpParam : "LFTP_typeFtpParam";
      instTconSettingsControl : TCONSettings;
      statTconSettingsControlReq : Bool;
      statTconSettingsControlOption : TCON_TCPTermination;   // Set TCP Termination for control connection to "Graceful shutdown"
      instTconControl : TCON;   // Tcon for FTP control connection
      statTconControlReq : Bool := FALSE;
      instTsendControl : TSEND;   // Tsend for FTP control commands
      statTsendControlReq : Bool := FALSE;
      statTsendControlLen : UInt;   // Length of data to be sent over control connection
      instTrcvControl : TRCV;   // Trcv for receiving reply codes from FTP-Server
      statTrcvControlEnable : Bool;   // Enable TRCV for control connection
      instTdisconControl : TDISCON;   // TDiscon for control connection
      statTdisconControlReq : Bool := FALSE;
      instTconSettingsData : TCONSettings;
      statTconSettingsDataReq : Bool;
      statTconSettingsDataOption : TCON_TCPTermination;   // Set TCP Termination for data connection to "Graceful shutdown"
      instTconData : TCON;   // Tcon for FTP data connection
      statTconDataReq : Bool := FALSE;
      instTsendData : TSEND;   // Tsend for sending data to FTP-Server
      statTsendDataReq : Bool := FALSE;
      instTrcvData : TRCV;   // Trcv for receiving data from the FTP-Server
      statTrcvDataEnable : Bool;   // Enable TRCV for data connection
      instTdisconData : TDISCON;   // TDiscon for data connection
      statTdisconDataReq : Bool := FALSE;
      statCtrlReplyCode : Int;   // Reply code received from FTP-Server
      statTsendControlData : Array[0..100] of Char;   // Data for Tsend of control connection
      statTrcvControlData : Array[0..149] of Char;   // Data for Trcv of data connection
      statTrcvControlString : String;
      statLocalHighPort : UInt;   // Local port (LowPort*256 + HighPort)
      statLocalLowPort : UInt;   // Local port (LowPort*256 + HighPort)
      statIpAsString : String;   // Client IP-Adress as a String
      statLocalPortAsString : String;   // Local Port combined as String
      statPortPosition : Int;
      statSearchPosition : Int;
      statRemotePortLowStr : String;   // Remote LowPort for passive mode as String (LowPort*256 + HighPort)
      statRemotePortHighStr : String;   // Remote HighPort for passive mode as String (LowPort*256 + HighPort)
      statRemotePort : UInt;   // Combined remote port for passive mode
      statRcvDataBuffer : Array[0..8191] of Byte;
      statDataLen : UDInt;
      statCtrlConnectionID : Word;   // Connection ID of the control connection
      statDataConnectionID : Word;   // Connection ID of the data connection
      statCtrlConnEstablished : Bool;
      statDataConnEstablished : Bool;
      statUserCredentials : Struct
         username : String;
         password : String;
      END_STRUCT;
      instTimeout : TON_TIME;
      statTimeoutIn : Bool;
      instRdRec : RDREC;
      statRdRecRecord : Struct
         blockType : UInt;
         blockLength : UInt;
         blockVersionHigh : USInt;
         blockVersionLow : USInt;
         data : Array[0..#REC_IP_MLEN] of Byte;
      END_STRUCT;
   END_VAR
   VAR_TEMP
      tempUrl : String;
      tempPos : Int;
      tempString : String;
      tempIndex : DInt;
      tempRet : Word;   // Return value
      tempStartIpAddress : USInt;   // Start of IP address in data record
   END_VAR
   VAR CONSTANT
      FB_STATE_NO_PROCESSING : UInt := 0;   // FB state: No processing
      FB_STATE_EVAL_CONN_PARAM : UInt := 10;   // FB state: Evaluate connection parameters
      FB_STATE_GET_ID_CTRL : UInt := 11;   // FB state: Get connection ID for control connection
      FB_STATE_EST_CTRL_CONN : UInt := 20;   // FB state: Establish control connection
      FB_STATE_SEND_USERNAME : UInt := 30;   // FB state: Send FTP username
      FB_STATE_USERNAME_SENT : UInt := 31;   // FB state: FTP username sent, wait for reply code 331
      FB_STATE_SEND_PASSWORD : UInt := 32;   // FB state: Send password
      FB_STATE_PASSWORD_SENT : UInt := 33;   // FB state: Password sent, wait for reply code 230
      FB_STATE_SET_CON_TYPE : UInt := 34;   // FB state: Set type of FTP connection ("Type I")
      FB_STATE_TYPE_SENT : UInt := 35;   // FB state: Type of FTP connection SENT
      FB_STATE_CTRL_CONN_EST : UInt := 50;   // FB state: Control connection established
      FB_STATE_GET_ID_DATA : UInt := 51;   // FB state: Get connection ID for data connection
      FB_STATE_GET_IP_INFO : UInt := 52;   // FB state: Get IP of PLC for FTP active mode
      FB_STATE_SEND_FTP_MODE : UInt := 53;   // FB state: Send FTP mode
      FB_STATE_EST_DATA_CONN : UInt := 54;   // FB state: FTP mode sent, establishing data connection
      FB_STATE_SEND_FILENAME_CMD : UInt := 55;   // FB state: Send filename and FTP-command
      FB_STATE_FILENAME_CMD_SENT : UInt := 56;   // FB state: Filename and command sent
      FB_STATE_DATA_TRANSFER : UInt := 60;   // FB state: Data transfer
      FB_STATE_CLOSE_DATA_CON : UInt := 70;   // FB state: Close data connection
      FB_STATE_SEND_QUIT : UInt := 90;   // FB state: Send 'Quit' command
      FB_STATE_DISCONNECT_CTRL : UInt := 91;   // FB state: Close control connection
      STATUS_EXECUTION_FINISHED : Word := 16#0000;   // Execution finished without errors
      STATUS_NO_CALL : Word := 16#7000;   // FB in idle, no active connection
      STATUS_FIRST_CALL : Word := 16#7001;   // First call after incoming new job (rising edge 'enable')
      STATUS_ESTABLISH_CTRL_CON : Word := 16#7002;   // Establish control connection
      STATUS_DISCON_CONTRL_CON : Word := 16#7003;   // Disconnect control connection
      STATUS_CONNECTED : Word := 16#7004;   // Control connection established
      STATUS_FTP_COMMAND_EXECUTE : Word := 16#7005;   // Execute selected FTP command
      ERR_TSEND_TERMINATED : Word := 16#80C5;   // TSEND: The remote partner has terminated the connection
      ERR_TRCV_TEMP_COMM_ERR : Word := 16#80C4;   // TRCV: Temporary communication error
      ERR_TRCV_TERMINATED : Word := 16#80C5;   // TRCV: The remote partner has terminated the connection.
      ERR_INVALID_URL : Word := 16#8202;   // Error: Invalid URL
      ERR_FROM_FTP_SERVER : Word := 16#8400;   // Error: Server sent an error reply code
      ERR_UNDEFINED_STATE : Word := 16#8600;   // Error: Due to an undefined state in state machine
      ERR_TCON : Word := 16#8601;   // Error: error on TCON
      ERR_TSEND : Word := 16#8602;   // Error: error on TSEND
      ERR_TRCV : Word := 16#8603;   // Error: error on TRCV
      ERR_TCONSETTINGS : Word := 16#8604;   // Error: error on TCONSETTINGS
      ERR_MOVE_BLK_VARIANT : Word := 16#8605;   // Error: error while move blk variant
      ERR_RDREC : Word := 16#8606;   // Error from RDREC
      ERR_WATCHDOG_TIMED_OUT : Word := 16#8DF1;   // Error: Action needs too long
      ERR_UNKNOWN_REPLY : Word := 16#8DF2;   // Error: Unknown replycode
      ERR_UNKNOWN_COMMAND : Word := 16#8DF3;   // Error: Unknown ftpcmd
      ERR_INVALID_ACTIVE_PORT : Word := 16#8DF4;   // Error: Port for active mode wrong
      SUB_STATUS_NO_ERROR : Word := 16#0000;   // No error occured in subfunction call
      PORT_FTP_DATA : UInt := 20;   // Remote port for FTP data connection
      PORT_FTP_CTRL : UInt := 21;   // Remote port for FTP control connection
      CONNECTION_TYPE_TCPIP : Byte := 16#0B;   // Connection Type set to TCP/IP
      CMD_STORE : Int := 2;   // FTP command "STOR"
      CMD_RETRIEVE : Int := 3;   // FTP command "RETR"
      CMD_DELETE : Int := 4;   // FTP command "DELE"
      CMD_APPEND : Int := 6;   // FTP command "APPE"
      REPLY_CODE_START_TRANSFER : Int := 150;   // Reply code: 150 "About to start data transfer"
      REPLY_CODE_200 : Int := 200;   // Reply code: 200 "Port command successful" or "Goodbye" or "Type set to I"
      REPLY_CODE_CONN_EST : Int := 220;   // Reply code: 220 server is ready for the client
      REPLY_CODE_QUIT_SENT : Int := 221;   // Reply code: 221 response to "QUIT" command
      REPLY_CODE_OP_SUCCESS : Int := 226;   // Reply code: 226 "Operation successful"
      REPLY_CODE_PASV_SUCCESS : Int := 227;   // Reply code: 227 "Entering Passive Mode (IP,LowPort,HighPort)"
      REPLY_CODE_PASSWORD_OK : Int := 230;   // Reply code: 230 "Login successful"
      REPLY_CODE_DELETE_SUCCESS : Int := 250;   // Reply code: 250 "File deleted successfully"
      REPLY_CODE_USERNAME_OK : Int := 331;   // Reply code: 331 "Please, specify the password"
      REPLY_CODE_ERROR_LOW : Int := 400;   // Reply code: 400, low end error reply codes from server
      REPLY_CODE_ERROR_HIGH : Int := 599;   // Reply code: 599, high end error reply codes from server
      REPLY_CODE_CONN_TIME_OUT : Int := 421;   // Reply code: 421 connection timed out
      REPLY_CODE_DATA_NOT_OPENED : Int := 425;   // Reply code: 425 could not open data connection
      REPLY_CODE_TRANSF_ABORTED : Int := 426;   // Reply code: 426 connection aborted, transfer aborted
      REPLY_CODE_ACTION_ABORTED : Int := 450;   // Reply code: 450 action aborted
      REPLY_CODE_SYNTAX_ERROR : Int := 500;   // Reply code: 500 syntax error
      REPLY_CODE_BAD_SEQUENCE : Int := 503;   // Reply code: 503 response to any command that requires the successful processing of previous commands first
      REPLY_CODE_NOT_LOGGED_IN : Int := 530;   // Reply code: 530 "Not logged in"
      REPLY_CODE_FILE_NOT_FOUND : Int := 550;   // Reply code: 550 filename not found, couldn´t open the file
      MSG_CONN_TYPE : String := 'TYPE I$R$L';   // Message connection type
      MSG_QUIT : String := 'QUIT$R$L';   // Message quit
      REC_IP_INDEX : DInt := 32896;   // Index of record PDInterfaceDataReal (0x8080)
      REC_IP_MLEN : UInt := 159;   // Maximum length of record PDInterfaceDataReal
      REC_LEN_BLOCK_HEADER : USInt := 6;   // Length of blocker header
      REC_LEN_NAME_LEN : USInt := 1;   // Length of station name length
      REC_LEN_MAC : USInt := 8;   // Length of MAC address in record PDInterfaceDataReal
   END_VAR
   // instTsendData.REQ := FALSE;
   // instTsendData.DONE := FALSE;
   // instTsendData.BUSY := FALSE;
   // instTsendData.ERROR := FALSE;
   // instTconControl.REQ := FALSE;
   // instTconControl.DONE := FALSE;
   // instTconControl.BUSY := FALSE;
   // instTconControl.ERROR := FALSE;
   // instTrcvData.ERROR := FALSE;
   // instTrcvControl.ADHOC := FALSE;
   // instTrcvControl.NDR := FALSE;
   // instTrcvControl.BUSY := FALSE;
   // instTrcvControl.ERROR := FALSE;
   // instTconData.REQ := FALSE;
   // instTconData.DONE := FALSE;
   // instTconData.BUSY := FALSE;
   // instTconData.ERROR := FALSE;
   // instTrcvData.EN_R := FALSE;
   // instTsendControl.REQ := FALSE;
   // instTsendControl.DONE := FALSE;
   // instTsendControl.BUSY := FALSE;
   // instTsendControl.ERROR := FALSE;
   // instTrcvControl.EN_R := FALSE;
   // instTrcvData.ADHOC := FALSE;
   // instTrcvData.NDR := FALSE;
   // instTrcvData.BUSY := FALSE;
   // statTconSettingsDataOption.GracefulShutdown := TRUE;
   // statTconSettingsControlOption.GracefulShutdown := TRUE;
BEGIN
   REGION BLOCK INFO HEADER
     //===============================================================================
     // SIEMENS / (c)Copyright 2022
     //-------------------------------------------------------------------------------
     // Title:            LFTP_Client
     // Function:         Implements an FTP client
     // Library:          LFTP
     // Author:           Siemens Industry Online Support
     // Tested with:      CPU 1513-1 PN FW 2.9
     //                   CPU 1215C FW 4.5
     // Engineering:      TIA Portal V17
     // Restrictions:     --
     // Requirements:     S7-1500 CPU with FW 2.9 or higher
     //                   S7-1200 CPU with FW 4.5 or higher
     // Change log table:
     // Version  | Date       | Expert in charge       | Changes applied
     //----------|------------|------------------------|------------------------------
     // 06.01.01 | 2023-04-14 | Online Support         | Fixed statSubfunctionStatus datatype bug (Problems with status from RdRec)
     //                                                | Word -> DWord
     //----------|------------|------------------------|------------------------------
     // 06.01.00 | 2022-11-14 | Online Support         | Replaced CommConfig with RDREC for compatibility with S7-1200
     //                                                | Fixed timeout bug
     //----------|------------|------------------------|------------------------------
     // 06.00.00 | 2022-05-30 | Online Support         | Complete code refactoring
     //                                                | Changed interface in accordance with PLCopen
     //                                                | Added automatic assignment of connection ID
     //                                                | Added parameter to specify length of data to be sent and output length of data received
     //                                                | Bug fixes
     //----------|------------|------------------------|------------------------------
     // 05.00.00 | 2021-02-01 | Online Support         | Upgrade to TIA Portal V16 Update 3
     //----------|------------|------------------------|------------------------------
     // 04.00.00 | 2019-07-01 | Online Support         | Upgrade to TIA Portal V15.1
     //----------|------------|------------------------|------------------------------
     // 03.05.00 | 2019-02-01 | Online Support         | Bug fixes
     //----------|------------|------------------------|------------------------------
     // 03.03.00 | 2018-03-01 | Online Support         | Upgrade to TIA Portal V15
     //                                                | Bug fixes
     //----------|------------|------------------------|------------------------------
     // 03.01.00 | 2017-11-01 | Online Support         | Bug fixes and performance improvements
     //----------|------------|------------------------|------------------------------
     // 03.00.00 | 2017-07-01 | Online Support         | Upgrade to TIA Portal V14 SP1
     //                                                | Complete revision of the "Ftp1X00Cmd" block according to the programming style guide
     //----------|------------|------------------------|------------------------------
     // 02.00.00 | 2015-05-01 | Online Support         | Upgrade to TIA Portal V13 SP1
     //                                                | Update of OUC blocks
     //----------|------------|------------------------|------------------------------
     // 01.00.00 | 2013-10-01 | Online Support         | First released version
     //===============================================================================
   END_REGION

   REGION ENABLING/DISABLING
     IF #enable AND #statStatus = #STATUS_NO_CALL THEN // Enable FB
       // First call; initialize FB
       #statValid := TRUE;
       #statDone := FALSE;
       #statBusy := TRUE;
       #statError := FALSE;
       #statErrorUserCleared := FALSE;
       #statErrorAutoCleared := FALSE;
       #statSubfunctionStatus := #SUB_STATUS_NO_ERROR;
       #statFBErrorState := 0;
       #diagnostics := #statEmptyDiagnostics;
       #statDisablingCompleted := FALSE;

       //Control Connection
       #statTconControlReq := FALSE;
       #statTdisconControlReq := FALSE;
       #statTconSettingsControlReq := FALSE;
       #statTsendControlReq := FALSE;
       #statTrcvControlEnable := FALSE;
       #statCtrlConnectionID := 0;

       //Data Connection
       #statTconDataReq := FALSE;
       #statTdisconDataReq := FALSE;
       #statTconSettingsDataReq := FALSE;
       #statTsendDataReq := FALSE;
       #statTrcvDataEnable := FALSE;

       // State machine - start functionality
       #statFBState := #FB_STATE_EVAL_CONN_PARAM;
       #statTimeoutIn := TRUE;
       RESET_TIMER(#instTimeout);
       #statStatus := #STATUS_FIRST_CALL;

     ELSIF NOT #enable AND #statEnableOld THEN // Disable FB
       #statDone := FALSE;
       #statErrorUserCleared := FALSE;
       #statErrorAutoCleared := FALSE;
       #statStatus := #STATUS_DISCON_CONTRL_CON;

       // Start and reset timer in case it was already running 
       #statTimeoutIn := TRUE;
       RESET_TIMER(#instTimeout);

       IF #statDataConnEstablished THEN // Data connection established
         #statFBState := #FB_STATE_CLOSE_DATA_CON;
       ELSIF #statCtrlConnEstablished THEN // Only control connection established 
         #statFBState := #FB_STATE_SEND_QUIT;
       ELSE // No connection established
         #statFBState := #FB_STATE_DISCONNECT_CTRL;
       END_IF;
     END_IF;

     // Edge detection
     #statEnableOld := #enable;
   END_REGION ENABLING/DISABLING

   IF (#statStatus = #STATUS_NO_CALL) THEN // Nothing to do -> End here to reduce "system load"
     RETURN;
   END_IF;

   REGION WATCHDOG
     // Monitor time out   
     #instTimeout(IN := #statTimeoutIn,
                  PT := #timeOut);

     IF #instTimeout.Q THEN
       #statTimeoutIn := FALSE;
       #statTconSettingsControlReq := FALSE;

       IF #statFBState = #FB_STATE_SEND_QUIT THEN
         #statFBState := #FB_STATE_DISCONNECT_CTRL; // Skip to disconnection
       ELSE
         #statStatus := #ERR_WATCHDOG_TIMED_OUT;
         #statFBErrorState := #statFBState;
         #statSubfunctionStatus := #SUB_STATUS_NO_ERROR;

         IF #statFBState >= #FB_STATE_CTRL_CONN_EST AND #statFBState < #FB_STATE_CLOSE_DATA_CON THEN // Timeout of FTP command
           #statErrorAutoCleared := TRUE;
           #statFBState := #FB_STATE_CLOSE_DATA_CON;
         ELSE
           #statErrorUserCleared := TRUE;
         END_IF;
       END_IF;
     END_IF;
   END_REGION

   REGION STATE_MACHINE  
     CASE #statFBState OF
       #FB_STATE_NO_PROCESSING:
         REGION no processing
           // No processing active (Note: this state must always be present and left empty)
           ;
         END_REGION no processing

       #FB_STATE_EVAL_CONN_PARAM..#FB_STATE_TYPE_SENT:
         REGION establish control connection

           CASE #statFBState OF
             #FB_STATE_EVAL_CONN_PARAM:
               REGION evaluate connection parameters
                 //QDN
                 #tempUrl := #connParam.serverAddress;
                 // Determine if host is domain name or IP address
                 #tempPos := CHAR_TO_INT(#tempUrl[1]);
                 IF #tempPos >= CHAR_TO_INT('A') AND #tempPos <= CHAR_TO_INT('z') THEN // Host is a domain name
                   #statConnParam.isQDN := true;
                 ELSIF #tempPos >= CHAR_TO_INT('0') AND #tempPos <= CHAR_TO_INT('9') THEN // Host is an IP address
                   #statConnParam.isQDN := false;
                 ELSE // URL invalid
                   #statStatus := #ERR_INVALID_URL;
                 END_IF;

                 IF #statConnParam.isQDN THEN // Host is a domain name
                   IF #tempUrl[LEN(#tempUrl)] = '.' THEN
                     #statConnParam.paramControlQDN.RemoteQDN := #tempUrl;
                   ELSE
                     #statConnParam.paramControlQDN.RemoteQDN := CONCAT(IN1 := #tempUrl, IN2 := '.');
                   END_IF;
                   #statConnParam.paramControlQDN.InterfaceId := #connParam.hwID;
                   #statConnParam.paramControlQDN.ConnectionType := #CONNECTION_TYPE_TCPIP;
                   #statConnParam.paramControlQDN.ActiveEstablished := TRUE;
                   #statConnParam.paramControlQDN.RemotePort := #PORT_FTP_CTRL;

                 ELSE // Host is an IP address
                   FOR #tempIndex := 1 TO 3 DO
                     #tempPos := FIND(IN1 := #tempUrl, IN2 := '.');
                     #statConnParam.paramControlIP.RemoteAddress.ADDR[#tempIndex] := UINT_TO_BYTE(STRING_TO_UINT(LEFT(IN := #tempUrl, L := #tempPos - 1)));
                     #tempUrl := DELETE(IN := #tempUrl, L := #tempPos, P := 1);
                   END_FOR;
                   #statConnParam.paramControlIP.RemoteAddress.ADDR[4] := UINT_TO_BYTE(STRING_TO_UINT(#tempUrl));
                   #statConnParam.paramControlIP.InterfaceId := #connParam.hwID;
                   #statConnParam.paramControlIP.ConnectionType := #CONNECTION_TYPE_TCPIP;
                   #statConnParam.paramControlIP.ActiveEstablished := TRUE;
                   #statConnParam.paramControlIP.RemotePort := #PORT_FTP_CTRL;
                 END_IF;

                 #statUserCredentials.username := #connParam.username;
                 #statUserCredentials.password := #connParam.password;

                 #statTconSettingsControlReq := TRUE;
                 #statFBState := #FB_STATE_GET_ID_CTRL;
               END_REGION

             #FB_STATE_GET_ID_CTRL:
               REGION get control connection ID
                 //Create Connection ID and Set TCP Termination to TCP Finish
                 IF #instTconSettingsControl.DONE THEN
                   #statTconSettingsControlReq := FALSE;
                   IF #statConnParam.isQDN THEN
                     #statConnParam.paramControlQDN.ID := #statCtrlConnectionID;
                   ELSE
                     #statConnParam.paramControlIP.ID := #statCtrlConnectionID;
                   END_IF;

                   #statTconControlReq := TRUE;
                   #statStatus := #STATUS_ESTABLISH_CTRL_CON;
                   #statFBState := #FB_STATE_EST_CTRL_CONN;
                 ELSIF #instTconSettingsControl.ERROR THEN
                   #statTconSettingsControlReq := FALSE;
                   #statErrorUserCleared := TRUE;
                   #statStatus := #ERR_TCONSETTINGS;
                   #statSubfunctionStatus := #instTconSettingsControl.STATUS;
                   #statFBErrorState := #statFBState;
                 END_IF;
               END_REGION

             #FB_STATE_EST_CTRL_CONN:
               REGION wait for Tcon ctrl conn DONE
                 //reset TCON Request
                 #statTconControlReq := FALSE;
                 //wait for reply code 220 of FTP server
                 IF #instTconControl.DONE THEN
                   #statCtrlConnEstablished := TRUE;
                   #statTrcvControlEnable := TRUE;
                 ELSIF #instTconControl.ERROR THEN
                   #statErrorUserCleared := TRUE;
                   #statStatus := #ERR_TCON;
                   #statSubfunctionStatus := #instTconControl.STATUS;
                   #statFBErrorState := #statFBState;
                 END_IF;
               END_REGION

             #FB_STATE_SEND_USERNAME:
               REGION send username
                 //Convert String to sendable array of chars
                 Strg_TO_Chars(Strg   := CONCAT(IN1 := 'USER ', IN2 := #statUserCredentials.username, IN3 := '$R$L'),
                               pChars := 0,
                               Cnt    => #statTsendControlLen,
                               Chars  := #statTsendControlData);

                 //send Username to FTP server
                 #statTsendControlReq := TRUE;
                 #statFBState := #FB_STATE_USERNAME_SENT;
               END_REGION

             #FB_STATE_USERNAME_SENT:
               //reply code 331 is expected
               #statTsendControlReq := FALSE;
               //wait for reply code of FTP server

               IF #instTsendControl.ERROR THEN
                 #statErrorUserCleared := TRUE;
                 #statStatus := #ERR_TSEND;
                 #statSubfunctionStatus := #instTsendControl.STATUS;
                 #statFBErrorState := #statFBState;
               END_IF;

             #FB_STATE_SEND_PASSWORD:
               REGION send password
                 //Convert String to sendable array of chars
                 Strg_TO_Chars(Strg   := CONCAT(IN1 := 'PASS ', IN2 := #statUserCredentials.password, IN3 := '$R$L'),
                               pChars := 0,
                               Cnt    => #statTsendControlLen,
                               Chars  := #statTsendControlData);

                 //send Password to FTP server
                 #statTsendControlReq := TRUE;
                 #statFBState := #FB_STATE_PASSWORD_SENT;
               END_REGION

             #FB_STATE_PASSWORD_SENT:
               //Password is sent, reply code 230 is expected
               #statTsendControlReq := FALSE;
               //wait for reply code 230 of FTP server

               IF #instTsendControl.ERROR THEN
                 #statErrorUserCleared := TRUE;
                 #statStatus := #ERR_TSEND;
                 #statSubfunctionStatus := #instTsendControl.STATUS;
                 #statFBErrorState := #statFBState;
               END_IF;

             #FB_STATE_SET_CON_TYPE:
               REGION set type of connection
                 //Convert String to sendable array of chars
                 Strg_TO_Chars(Strg   := #MSG_CONN_TYPE,
                               pChars := 0,
                               Cnt    => #statTsendControlLen,
                               Chars  := #statTsendControlData);

                 //send Type to FTP server
                 #statTsendControlReq := TRUE;
                 #statFBState := #FB_STATE_TYPE_SENT;
               END_REGION

             #FB_STATE_TYPE_SENT:
               //reply code 200 is expected
               #statTsendControlReq := FALSE;
               //wait for reply code 200 of FTP server

               IF #instTsendControl.ERROR THEN
                 #statErrorUserCleared := TRUE;
                 #statStatus := #ERR_TSEND;
                 #statSubfunctionStatus := #instTsendControl.STATUS;
                 #statFBErrorState := #statFBState;
               END_IF;

           END_CASE;
         END_REGION establish control connection

       #FB_STATE_CTRL_CONN_EST..#FB_STATE_CLOSE_DATA_CON:
         REGION control connection established

           CASE #statFBState OF
             #FB_STATE_CTRL_CONN_EST:
               //FTP commands could be executed now
               #statTimeoutIn := FALSE;

               IF #statStatus = #STATUS_ESTABLISH_CTRL_CON THEN
                 #statStatus := #STATUS_CONNECTED;
               END_IF;

               //FTP commands could be executed now
               REGION execute
                 IF #execute AND NOT #statExecuteOld THEN
                   #statDataConnectionID := 0;
                   // Save FTP parameters
                   #statFtpParam := #ftpParam;

                   //Check if FtpCmd is valid
                   IF #statFtpParam.ftpCmd = #CMD_STORE OR #statFtpParam.ftpCmd = #CMD_RETRIEVE OR #statFtpParam.ftpCmd = #CMD_APPEND OR #statFtpParam.ftpCmd = #CMD_DELETE THEN
                     // Check FTP mode
                     IF NOT #statFtpParam.ftpActiveMode OR (#statFtpParam.ftpActiveMode AND #statFtpParam.portActiveMode > 2000) THEN
                       #statTimeoutIn := TRUE;
                       #statStatus := #STATUS_FTP_COMMAND_EXECUTE;

                       IF #statFtpParam.ftpCmd = #CMD_DELETE THEN
                         #statFBState := #FB_STATE_SEND_FILENAME_CMD;
                       ELSE // STORE, APPEND, RETRIEVE
                         IF #statFtpParam.ftpCmd = #CMD_RETRIEVE THEN
                           #statDataLen := 0;
                         ELSE
                           #statDataLen := #dataLen;
                         END_IF;

                         // establish data connection
                         #statTconSettingsDataReq := TRUE;
                         #statFBState := #FB_STATE_GET_ID_DATA;
                       END_IF;

                     ELSE
                       //wrong port for active mode
                       #statErrorAutoCleared := TRUE;
                       #statStatus := #ERR_INVALID_ACTIVE_PORT;
                       #statSubfunctionStatus := #SUB_STATUS_NO_ERROR;
                       #statFBErrorState := #statFBState;
                     END_IF;

                   ELSE
                     //wrong command / unknown CMD 
                     #statErrorAutoCleared := TRUE;
                     #statStatus := #ERR_UNKNOWN_COMMAND;
                     #statSubfunctionStatus := #SUB_STATUS_NO_ERROR;
                     #statFBErrorState := #statFBState;
                   END_IF;

                 ELSIF NOT #execute AND (#statDone OR #statError) THEN // Execute reset
                   #statDone := FALSE;
                   #statErrorAutoCleared := FALSE;
                   #statCtrlReplyCode := 0;
                   #statStatus := #STATUS_CONNECTED;

                 END_IF; // execute triggered

                 // Edge detection
                 #statExecuteOld := #execute;
               END_REGION

             #FB_STATE_GET_ID_DATA:
               REGION get data connection ID
                 IF #instTconSettingsData.DONE THEN
                   #statTconSettingsDataReq := FALSE;

                   IF #ftpParam.ftpActiveMode AND #statIpAsString = '' THEN // Switch state depending of FTP mode
                     #statFBState := #FB_STATE_GET_IP_INFO;
                   ELSE
                     #statFBState := #FB_STATE_SEND_FTP_MODE;
                   END_IF;

                 ELSIF #instTconSettingsData.ERROR THEN
                   #statTconSettingsDataReq := FALSE;
                   #statErrorAutoCleared := TRUE;
                   #statStatus := #ERR_TCONSETTINGS;
                   #statSubfunctionStatus := #instTconSettingsData.STATUS;
                   #statFBErrorState := #statFBState;
                   #statFBState := #FB_STATE_CTRL_CONN_EST;
                 END_IF;
               END_REGION

             #FB_STATE_GET_IP_INFO:
               REGION get IP address for active mode

                 #instRdRec(REQ    := TRUE,
                            ID     := #connParam.hwID,
                            INDEX  := #REC_IP_INDEX,
                            MLEN   := #REC_IP_MLEN + 1,
                            RECORD := #statRdRecRecord);

                 IF #instRdRec.VALID OR #instRdRec.ERROR THEN
                   IF #instRdRec.VALID THEN
                     // Calculate start of IP address in data record
                     // Block header + length of station name + station name is padded to make them Unsigned32 aligned
                     #tempStartIpAddress := #REC_LEN_NAME_LEN + BYTE_TO_USINT(#statRdRecRecord.data[0]) + (4 - (#REC_LEN_BLOCK_HEADER + #REC_LEN_NAME_LEN + BYTE_TO_USINT(#statRdRecRecord.data[0])) MOD 4) MOD 4 + #REC_LEN_MAC;

                     // Convert IP address to String
                     #statIpAsString := DELETE(IN := UINT_TO_STRING(BYTE_TO_UINT(#statRdRecRecord.data[#tempStartIpAddress])), L := 1, P := 1);
                     #statIpAsString := CONCAT(IN1 := #statIpAsString, IN2 := ',');
                     #statIpAsString := CONCAT(IN1 := #statIpAsString, IN2 := DELETE(IN := UINT_TO_STRING(BYTE_TO_UINT(#statRdRecRecord.data[#tempStartIpAddress + 1])), L := 1, P := 1));
                     #statIpAsString := CONCAT(IN1 := #statIpAsString, IN2 := ',');
                     #statIpAsString := CONCAT(IN1 := #statIpAsString, IN2 := DELETE(IN := UINT_TO_STRING(BYTE_TO_UINT(#statRdRecRecord.data[#tempStartIpAddress + 2])), L := 1, P := 1));
                     #statIpAsString := CONCAT(IN1 := #statIpAsString, IN2 := ',');
                     #statIpAsString := CONCAT(IN1 := #statIpAsString, IN2 := DELETE(IN := UINT_TO_STRING(BYTE_TO_UINT(#statRdRecRecord.data[#tempStartIpAddress + 3])), L := 1, P := 1));
                     #statIpAsString := CONCAT(IN1 := #statIpAsString, IN2 := ',');

                     #statFBState := #FB_STATE_SEND_FTP_MODE;

                   ELSIF #instRdRec.ERROR THEN
                     #statErrorAutoCleared := TRUE;
                     #statStatus := #ERR_RDREC;
                     #statSubfunctionStatus := #instRdRec.STATUS;
                     #statFBErrorState := #statFBState;
                     #statFBState := #FB_STATE_CTRL_CONN_EST;
                   END_IF;

                   // Reset RDREC
                   #instRdRec(REQ    := FALSE,
                              RECORD := #statRdRecRecord);
                 END_IF;
               END_REGION

             #FB_STATE_SEND_FTP_MODE:
               REGION send FTP mode
                 // Parameters independent of FTP mode
                 IF #statConnParam.isQDN THEN //Remote adress is QDN
                   #statConnParam.paramDataQDN.InterfaceId := #connParam.hwID;
                   #statConnParam.paramDataQDN.ID := #statDataConnectionID;
                   #statConnParam.paramDataQDN.RemoteQDN := #statConnParam.paramControlQDN.RemoteQDN;
                 ELSE //Remote adress is IP address
                   #statConnParam.paramDataIP.InterfaceId := #connParam.hwID;
                   #statConnParam.paramDataIP.ID := #statDataConnectionID;
                   #statConnParam.paramDataIP.RemoteAddress := #statConnParam.paramControlIP.RemoteAddress;
                 END_IF;

                 // Parameters dependent of FTP mode
                 IF #ftpParam.ftpActiveMode THEN // Active FTP
                   //preparation for data connection in active mode (Connection ID Data and ID Control are generated by TCONSettings every time)
                   IF #statConnParam.isQDN THEN //Remote adress is QDN
                     #statConnParam.paramDataQDN.ActiveEstablished := FALSE;
                     #statConnParam.paramDataQDN.RemotePort := 0; // Accept any port
                     #statConnParam.paramDataQDN.LocalPort := #ftpParam.portActiveMode;
                   ELSE //Remote adress is IP address
                     #statConnParam.paramDataIP.ActiveEstablished := FALSE;
                     #statConnParam.paramDataIP.RemotePort := 0; // Accept any port
                     #statConnParam.paramDataIP.LocalPort := #ftpParam.portActiveMode;
                   END_IF;

                   //delete '+' signs out of Port String
                   //split local port to needed high and low port with formula PORT:=high*256+low
                   IF #statConnParam.isQDN THEN
                     #statLocalLowPort := #statConnParam.paramDataQDN.LocalPort MOD 256;
                     #statLocalHighPort := (#statConnParam.paramDataQDN.LocalPort - #statLocalLowPort) / 256;
                   ELSE
                     #statLocalLowPort := #statConnParam.paramDataIP.LocalPort MOD 256;
                     #statLocalHighPort := (#statConnParam.paramDataIP.LocalPort - #statLocalLowPort) / 256;
                   END_IF;

                   #statLocalPortAsString := CONCAT(IN1 := DELETE(IN := UINT_TO_STRING(#statLocalHighPort), L := 1, P := 1), IN2 := ',');
                   #statLocalPortAsString := CONCAT(IN1 := #statLocalPortAsString, IN2 := DELETE(IN := UINT_TO_STRING(#statLocalLowPort), L := 1, P := 1));

                   #tempString := CONCAT(IN1 := 'PORT ', IN2 := #statIpAsString, IN3 := #statLocalPortAsString, IN4 := '$R$L');

                   #statTconDataReq := TRUE; // In FTP active mode, port is opened right away

                 ELSE // Passive FTP
                   IF #statConnParam.isQDN THEN //Remote adress is QDN
                     //preparation for data connection in passive mode (ID Data and ID Control are generated by TCONSettings every time)
                     #statConnParam.paramDataQDN.ActiveEstablished := TRUE;
                     #statConnParam.paramDataQDN.LocalPort := 0; // Irrelevant
                   ELSE //Remote adress is IP address
                     //preparation for data connection in passive mode (ID Data and ID Control are generated by TCONSettings every time)
                     #statConnParam.paramDataIP.ActiveEstablished := TRUE;
                     #statConnParam.paramDataIP.LocalPort := 0; // Irrelevant
                   END_IF;

                   #tempString := CONCAT(IN1 := 'PASV ', IN2 := '$R$L');
                 END_IF;//ftp mode

                 Strg_TO_Chars(Strg   := #tempString,
                               pChars := 0,
                               Cnt    => #statTsendControlLen,
                               Chars  := #statTsendControlData);

                 #statTsendControlReq := TRUE;
                 #statFBState := #FB_STATE_EST_DATA_CONN;
               END_REGION

             #FB_STATE_EST_DATA_CONN:
               REGION establishing data connection
                 #statTsendControlReq := FALSE;
                 //Waiting for Reply code 227 (passive) or 200 (active) next step, when reaches the expected ftp reply codes

                 IF #instTconData.DONE THEN // In active mode, reply code moves state machine; in passive mode, wait for TCON to establish connection
                   #statDataConnEstablished := TRUE;
                   #statFBState := #FB_STATE_SEND_FILENAME_CMD;
                 ELSIF #instTconData.ERROR THEN
                   #statErrorUserCleared := TRUE;
                   #statStatus := #ERR_TCON;
                   #statSubfunctionStatus := #instTconData.STATUS;
                   #statFBErrorState := #statFBState;
                 END_IF;

                 IF #instTsendControl.ERROR THEN
                   #statErrorAutoCleared := TRUE;
                   #statStatus := #ERR_TSEND;
                   #statSubfunctionStatus := #instTsendControl.STATUS;
                   #statFBErrorState := #statFBState;
                   #statFBState := #FB_STATE_CLOSE_DATA_CON;
                 END_IF;
               END_REGION

             #FB_STATE_SEND_FILENAME_CMD:
               REGION send file name and command
                 #statTconDataReq := FALSE;

                 //send filename and command to the ftp server
                 CASE #ftpParam.ftpCmd OF
                   #CMD_STORE:
                     #tempString := CONCAT(IN1 := 'STOR ', IN2 := #ftpParam.filename, IN3 := '$R$L');
                   #CMD_RETRIEVE:
                     #tempString := CONCAT(IN1 := 'RETR ', IN2 := #ftpParam.filename, IN3 := '$R$L');
                   #CMD_DELETE:
                     #tempString := CONCAT(IN1 := 'DELE ', IN2 := #ftpParam.filename, IN3 := '$R$L');
                   #CMD_APPEND:
                     #tempString := CONCAT(IN1 := 'APPE ', IN2 := #ftpParam.filename, IN3 := '$R$L');
                 END_CASE;

                 //copy needed data to the send data of control connection
                 Strg_TO_Chars(Strg   := #tempString,
                               pChars := 0,
                               Cnt    => #statTsendControlLen,
                               Chars  := #statTsendControlData);

                 #statTsendControlReq := TRUE;
                 #statFBState := #FB_STATE_FILENAME_CMD_SENT;
               END_REGION send file name and command

             #FB_STATE_FILENAME_CMD_SENT:
               REGION file name and command sent
                 #statTsendControlReq := FALSE;
                 //wait for ftp reply code 150

                 IF #instTsendControl.ERROR THEN
                   #statErrorAutoCleared := TRUE;
                   #statStatus := #ERR_TSEND;
                   #statSubfunctionStatus := #instTsendControl.STATUS;
                   #statFBErrorState := #statFBState;
                   IF #statDataConnEstablished THEN // DELETE doesn't need data connection; state machine is moved by reply code
                     #statFBState := #FB_STATE_CLOSE_DATA_CON;
                   END_IF;
                 END_IF;
               END_REGION

             #FB_STATE_DATA_TRANSFER:
               REGION data transfer
                 CASE #ftpParam.ftpCmd OF
                   #CMD_STORE, #CMD_APPEND:
                     #statTsendDataReq := TRUE;

                     IF #instTsendData.DONE THEN
                       #statTsendDataReq := FALSE;
                       #statFBState := #FB_STATE_CLOSE_DATA_CON;
                     END_IF;

                   #CMD_RETRIEVE:
                     #statTrcvDataEnable := TRUE;

                     //if more than 8192 Bytes should be recieved data has to be buffered
                     IF #instTrcvData.NDR AND #instTrcvData.RCVD_LEN > 0 THEN
                       //copy Buffer to output
                       #tempRet := INT_TO_WORD(MOVE_BLK_VARIANT(SRC := #statRcvDataBuffer,
                                                                                        SRC_INDEX := 0,
                                                                                        COUNT := #instTrcvData.RCVD_LEN,
                                                                                        DEST => #data,
                                                                                        DEST_INDEX := UDINT_TO_DINT(#statDataLen)));

                       //the offset of data copying has to be set up to last rcvdLen
                       #statDataLen := #statDataLen + #instTrcvData.RCVD_LEN;

                       IF #tempRet <> 0 THEN
                         //Error while copying recieved data to the data array
                         #statErrorAutoCleared := TRUE;
                         #statStatus := #ERR_MOVE_BLK_VARIANT;
                         #statSubfunctionStatus := #tempRet;
                         #statFBErrorState := #statFBState;
                         #statFBState := #FB_STATE_CLOSE_DATA_CON;
                       END_IF;

                     ELSIF #statCtrlReplyCode = #REPLY_CODE_OP_SUCCESS // Server sent reply code successful
                       AND #instTrcvData.ERROR AND (#instTrcvData.STATUS = #ERR_TRCV_TEMP_COMM_ERR OR #instTrcvData.STATUS = #ERR_TRCV_TERMINATED) // and connection was terminated
                     THEN
                       #statFBState := #FB_STATE_CLOSE_DATA_CON;

                     ELSIF #instTrcvData.ERROR AND NOT (#instTrcvData.STATUS = #ERR_TRCV_TEMP_COMM_ERR OR #instTrcvData.STATUS = #ERR_TRCV_TERMINATED) THEN
                       #statErrorAutoCleared := TRUE;
                       #statStatus := #ERR_TRCV;
                       #statSubfunctionStatus := #instTrcvData.STATUS;
                       #statFBErrorState := #statFBState;
                       #statFBState := #FB_STATE_CLOSE_DATA_CON;
                     END_IF;

                 END_CASE;
               END_REGION data transfer

             #FB_STATE_CLOSE_DATA_CON: //Close data connection
               REGION close data connection         
                 #statTrcvDataEnable := FALSE;
                 #statTdisconDataReq := TRUE;

                 //data channel has been closed
                 IF (#instTdisconData.DONE OR #instTdisconData.ERROR) THEN
                   #statTdisconDataReq := FALSE;
                   #statDataConnEstablished := FALSE;
                   #statTimeoutIn := FALSE;

                   IF #enable THEN // FB is enabled
                     #statFBState := #FB_STATE_CTRL_CONN_EST;

                     IF #statCtrlReplyCode < #REPLY_CODE_ERROR_LOW AND NOT #statError THEN // Success
                       #statDone := TRUE;
                       #statStatus := #STATUS_EXECUTION_FINISHED;
                     END_IF;

                   ELSE // Disabling
                     #statFBState := #FB_STATE_SEND_QUIT;
                   END_IF;
                 END_IF;
               END_REGION close data connection
           END_CASE; // Case for ftp data connection
         END_REGION control connection established

       #FB_STATE_SEND_QUIT:
         REGION send quit
           Strg_TO_Chars(Strg   := #MSG_QUIT,
                         pChars := 0,
                         Cnt    => #statTsendControlLen,
                         Chars  := #statTsendControlData);

           #statTsendControlReq := TRUE;

           IF #instTsendControl.ERROR AND NOT #instTsendControl.STATUS = #ERR_TSEND_TERMINATED THEN
             #statErrorAutoCleared := TRUE;
             #statStatus := #ERR_TSEND;
             #statSubfunctionStatus := #instTsendControl.STATUS;
             #statFBErrorState := #statFBState;
             #statFBState := #FB_STATE_DISCONNECT_CTRL;
           END_IF;
         END_REGION send quit

       #FB_STATE_DISCONNECT_CTRL:
         REGION disconnect connections
           #statTsendControlReq := FALSE;
           #statTrcvControlEnable := FALSE;
           #statTdisconControlReq := TRUE;

           IF #instTdisconControl.DONE OR #instTdisconControl.ERROR THEN // Don't wait for termination of data connection
             #statTdisconControlReq := FALSE;
             #statCtrlConnEstablished := FALSE;
             #statTimeoutIn := FALSE;
             #statDisablingCompleted := TRUE;
             #statFBState := #FB_STATE_NO_PROCESSING;
           END_IF;
         END_REGION disconnect connections

       ELSE // Undefined state in state machine reached
         REGION undefined state        
           #statStatus := #ERR_UNDEFINED_STATE;
           #statErrorUserCleared := TRUE;
         END_REGION undefined state

     END_CASE; // statemachine
   END_REGION STATE_MACHINE

   REGION OUC blocks control connection
     IF #statFBState <> #FB_STATE_NO_PROCESSING THEN // Only execute when FB is active to reduce system load
       IF #statConnParam.isQDN THEN // url is QDN
         #instTconControl(REQ     := #statTconControlReq,
                          ID      := #statConnParam.paramControlQDN.ID,
                          CONNECT := #statConnParam.paramControlQDN);
       ELSE // url is IP address
         #instTconControl(REQ     := #statTconControlReq,
                          ID      := #statConnParam.paramControlIP.ID,
                          CONNECT := #statConnParam.paramControlIP);
       END_IF;

       #instTconSettingsControl(REQ    := #statTconSettingsControlReq,
                                MODE   := 0,
                                ID     := #statCtrlConnectionID,
                                OPTION := #statTconSettingsControlOption);

       #instTrcvControl(EN_R  := #statTrcvControlEnable,
                        ID    := #statCtrlConnectionID,
                        LEN   := 0,
                        ADHOC := TRUE,
                        DATA  := #statTrcvControlData);

       #instTsendControl(REQ  := #statTsendControlReq,
                         ID   := #statCtrlConnectionID,
                         LEN  := #statTsendControlLen,
                         DATA := #statTsendControlData);

       #instTdisconControl(REQ := #statTdisconControlReq,
                           ID  := #statCtrlConnectionID);

       IF #instTrcvControl.ERROR THEN
         #statErrorUserCleared := TRUE;
         #statStatus := #ERR_TRCV;
         #statSubfunctionStatus := #instTrcvControl.STATUS;
         #statFBErrorState := #statFBState;

         // Connection disturbed
         IF #instTrcvControl.STATUS = #ERR_TRCV_TEMP_COMM_ERR
           OR #instTrcvControl.STATUS = #ERR_TRCV_TERMINATED
         THEN
           #statCtrlConnEstablished := FALSE;
         END_IF;
       END_IF;
     END_IF;
   END_REGION OUC blocks control connection

   REGION OUC blocks data connection
     IF (#statFBState <> #FB_STATE_NO_PROCESSING) THEN // Only execute when FB is active to reduce system load
       IF #statConnParam.isQDN THEN //url is QDN
         #instTconData(REQ     := #statTconDataReq,
                       ID      := #statConnParam.paramDataQDN.ID,
                       CONNECT := #statConnParam.paramDataQDN);
       ELSE //url is IP address
         #instTconData(REQ     := #statTconDataReq,
                       ID      := #statConnParam.paramDataIP.ID,
                       CONNECT := #statConnParam.paramDataIP);
       END_IF;

       #instTconSettingsData(REQ    := #statTconSettingsDataReq,
                             MODE   := 0,
                             ID     := #statDataConnectionID,
                             OPTION := #statTconSettingsDataOption);

       #instTrcvData(EN_R  := #statTrcvDataEnable,
                     ID    := #statDataConnectionID,
                     LEN   := 0,
                     ADHOC := TRUE,
                     DATA  := #statRcvDataBuffer);

       #instTsendData(REQ  := #statTsendDataReq,
                      ID   := #statDataConnectionID,
                      LEN  := #statDataLen,
                      DATA := #data);

       #instTdisconData(REQ := #statTdisconDataReq,
                        ID  := #statDataConnectionID);
     END_IF;
   END_REGION OUC blocks data connection

   REGION Eval FTP reply codes
     IF #instTrcvControl.NDR THEN
       // Extract reply code
       Chars_TO_Strg(Chars  := #statTrcvControlData,
                     pChars := 0,
                     Cnt    := 3,
                     Strg   => #statTrcvControlString);

       IF STRING_TO_INT(#statTrcvControlString) <> 0 THEN
         #statCtrlReplyCode := STRING_TO_INT(#statTrcvControlString);
       END_IF;

       //Check for all reply codes and send to the right step
       CASE #statCtrlReplyCode OF
         #REPLY_CODE_START_TRANSFER:
           //file status okay, about to open data connection
           //reset TSEND.REQ of Control connection
           #statTsendControlReq := FALSE;
           #statFBState := #FB_STATE_DATA_TRANSFER;

         #REPLY_CODE_200: // Port command successful, Goodbye or Type set to I
           IF #statFBState = #FB_STATE_SEND_QUIT OR #statFBState = #FB_STATE_DISCONNECT_CTRL THEN // Response Goodbye
             #statFBState := #FB_STATE_DISCONNECT_CTRL;
           ELSIF #statFBState >= #FB_STATE_TYPE_SENT AND #statFBState < #FB_STATE_SEND_FTP_MODE THEN
             //Type sent successfully
             //Connection and authentification were successfull, now idle and wait for new commands
             #statFBState := #FB_STATE_CTRL_CONN_EST;
           ELSE
             //Active is set successfully
             //PORT cmd was successful -> open data connection, so its open for communication with ftp server
             #statDataConnEstablished := TRUE;
             #statFBState := #FB_STATE_SEND_FILENAME_CMD;
           END_IF;

         #REPLY_CODE_CONN_EST:
           IF #statFBState < #FB_STATE_SEND_QUIT THEN
             #statFBState := #FB_STATE_SEND_USERNAME;
           END_IF;

         #REPLY_CODE_QUIT_SENT:
           #statFBState := #FB_STATE_DISCONNECT_CTRL;

         #REPLY_CODE_OP_SUCCESS:
           ; // Reply code is evaluated within state machine

         #REPLY_CODE_PASV_SUCCESS:
           //Server sent PORT -> it has to be found in received data of control connections TRCV
           //search FOR ')' because ftp Server sends: (IP1,IP2,IP3,IP4,PORT High,PORT Low)
           #statPortPosition := 0;
           #statRemotePortLowStr := '';
           #statRemotePortHighStr := '';

           FOR #statSearchPosition := 0 TO UDINT_TO_INT(#instTrcvControl.RCVD_LEN) - 1 DO
             IF #statTrcvControlData[#statSearchPosition] = ')' THEN
               #statPortPosition := #statSearchPosition;
             END_IF;
           END_FOR;
           //')' found -> search port 
           IF #statPortPosition > 0 THEN
             #statPortPosition := #statPortPosition - 1; //start with first sign before ')'
             WHILE #statTrcvControlData[#statPortPosition] <> ',' DO
               #statRemotePortLowStr := CONCAT(IN1 := #statTrcvControlData[#statPortPosition], IN2 := #statRemotePortLowStr);
               #statPortPosition := #statPortPosition - 1;
             END_WHILE;
             #statPortPosition := #statPortPosition - 1; //ongoing one position before ','
             WHILE #statTrcvControlData[#statPortPosition] <> ',' DO
               #statRemotePortHighStr := CONCAT(IN1 := #statTrcvControlData[#statPortPosition], IN2 := #statRemotePortHighStr);
               #statPortPosition := #statPortPosition - 1;
             END_WHILE;
             //calculation for Remote Port
             //remote port = high port * 256 + low port 
             #statRemotePort := STRING_TO_UINT(IN := #statRemotePortHighStr) * 256 + STRING_TO_UINT(#statRemotePortLowStr);
             #statConnParam.paramDataIP.RemotePort := #statRemotePort;
           END_IF; //statPortPositions > 0

           #statTconDataReq := TRUE;

         #REPLY_CODE_PASSWORD_OK:
           #statFBState := #FB_STATE_SET_CON_TYPE; //statStep 70

         #REPLY_CODE_DELETE_SUCCESS:
           #statTsendControlReq := FALSE;
           #statDone := TRUE;
           #statStatus := #STATUS_EXECUTION_FINISHED;
           #statFBState := #FB_STATE_CTRL_CONN_EST;

         #REPLY_CODE_USERNAME_OK:
           #statFBState := #FB_STATE_SEND_PASSWORD; //statStep 50

         #REPLY_CODE_ERROR_LOW..#REPLY_CODE_ERROR_HIGH: // Error
           #statTimeoutIn := FALSE;
           #statTconDataReq := FALSE;
           #statStatus := #ERR_FROM_FTP_SERVER;
           #tempRet := ATH(IN := #statTrcvControlString, N := 3, OUT => #statSubfunctionStatus); // Interpret response code as hexadecimal
           #statSubfunctionStatus := SHR(IN := #statSubfunctionStatus, N := 4);

           #statFBErrorState := #statFBState;

           CASE #statCtrlReplyCode OF // Error reply codes
             #REPLY_CODE_CONN_TIME_OUT:
               #statErrorUserCleared := TRUE;

             #REPLY_CODE_DATA_NOT_OPENED:
               #statErrorAutoCleared := TRUE;
               #statFBState := #FB_STATE_CLOSE_DATA_CON;

             #REPLY_CODE_TRANSF_ABORTED:
               #statErrorAutoCleared := TRUE;
               #statFBState := #FB_STATE_CLOSE_DATA_CON;

             #REPLY_CODE_ACTION_ABORTED:
               #statErrorAutoCleared := TRUE;
               #statFBState := #FB_STATE_CLOSE_DATA_CON;

             #REPLY_CODE_SYNTAX_ERROR:
               //Syntax Error, FB is not working correctly
               ;

             #REPLY_CODE_BAD_SEQUENCE:
               //ftp connection has to be reseted control and data connection have to be closed
               #statErrorAutoCleared := TRUE;
               #statFBState := #FB_STATE_CLOSE_DATA_CON;

             #REPLY_CODE_NOT_LOGGED_IN:
               #statErrorUserCleared := TRUE;

             #REPLY_CODE_FILE_NOT_FOUND:
               #statErrorAutoCleared := TRUE;
               #statTsendControlReq := FALSE;
               #statFBState := #FB_STATE_CLOSE_DATA_CON;
           END_CASE; // Error reply codes

         ELSE // unknown reply code
           #statTconDataReq := FALSE;
           #statTsendControlReq := FALSE;
           #statErrorUserCleared := TRUE;
           #statFBState := #FB_STATE_CLOSE_DATA_CON;
           #statStatus := #ERR_UNKNOWN_REPLY; //unknown reply code
           #statSubfunctionStatus := INT_TO_WORD(#statCtrlReplyCode);

       END_CASE; // Reply codes
     END_IF;
   END_REGION

   REGION OUTPUTS
     IF (#statDisablingCompleted) THEN
       REGION disabling completed
         #statValid := FALSE;
         #statDone := FALSE;
         #statError := FALSE;
         #statBusy := FALSE;
         #statStatus := #STATUS_NO_CALL;
         #statErrorUserCleared := FALSE;
         #statErrorAutoCleared := FALSE;
       END_REGION

     ELSIF (#statErrorUserCleared = TRUE) AND (#statError = FALSE) THEN
       REGION error user cleared
         // Error can only be cleared by user; rising edge at enable input is needed to continue 
         #statValid := FALSE;
         #statBusy := FALSE;
         #statError := TRUE;
         #statTimeoutIn := FALSE;
         // Write diagnostics
         #diagnostics.status := #statStatus;
         #diagnostics.subfunctionStatus := #statSubfunctionStatus;
         #diagnostics.stateNumber := #statFBErrorState;
         // execution aborted --> set state no processing
         #statFBState := #FB_STATE_NO_PROCESSING;
       END_REGION error user cleared

     ELSIF (#statErrorAutoCleared = TRUE) AND (#statError = FALSE) THEN
       REGION error auto cleared
         // Error can be reset by FB automatically
         #statValid := FALSE;
         #statBusy := TRUE;
         #statError := TRUE;
         #statTimeoutIn := FALSE;
         // Write diagnostics
         #diagnostics.status := #statStatus;
         #diagnostics.subfunctionStatus := #statSubfunctionStatus;
         #diagnostics.stateNumber := #statFBErrorState;
       END_REGION error auto cleared

     ELSIF (#statErrorAutoCleared = FALSE) AND (#statErrorUserCleared = FALSE) AND (#statError = TRUE) THEN
       REGION after user/auto cleared
         // If autocleared error is acknowledged
         #statValid := TRUE;
         #statBusy := TRUE;
         #statError := FALSE;
       END_REGION after user/auto cleared
     END_IF;

     REGION write static values to outputs
       #done := #statDone;
       #busy := #statBusy;
       #error := #statError;
       #valid := #statValid;
       #status := #statStatus;

       // Output received length
       IF #statDone AND #statFtpParam.ftpCmd = #CMD_RETRIEVE THEN
         #dataLen := #statDataLen;
       END_IF;
     END_REGION write static values to outputs
   END_REGION OUTPUTS
END_FUNCTION_BLOCK

(* ===== HMI "HMI_RT_1" =====
system functions are stored by id; their names below are inferred from use
connection "HMI_Connection_1": ETHERNET, S7_1200_OMS

HMI tags "Default tag table"
   "Tag_ScreenNumber" : USInt = PLC HMI_screen_no AT %MB96, 1 s
   "HMI_Tag_temp_login" : WString[254], internal
   "HMI_Tag_temp_password" : WString[254], internal
   "HMI_Tag_1_temp_user_number" : Int, internal
   "HMI_Tag_1" : Int, internal
   "V_zadane" : Int = PLC V_zadane AT %MW88, 1 s
   "V_zmierzone" : Int = PLC V_zmierzone AT %MW92, 1 s

HMI tags "Recipes_tags"
   "HMI_Tag_T1" : Int = PLC Recipe_db.Time_array[0] AT %MW40, 1 s
   "HMI_Tag_T2" : Int = PLC Recipe_db.Time_array[1] AT %MW44, 1 s
   "HMI_Tag_T3" : Int = PLC Recipe_db.Time_array[2] AT %MW48, 1 s
   "HMI_Tag_T4" : Int = PLC Recipe_db.Time_array[3] AT %MW52, 1 s
   "HMI_Tag_T5" : Int = PLC Recipe_db.Time_array[4] AT %MW56, 1 s
   "HMI_Tag_T6" : Int = PLC Recipe_db.Time_array[5] AT %MW60, 1 s
   "HMI_Tag_V1" : Int = PLC Recipe_db.Velocity_array[0] AT %MW64, 1 s
   "HMI_Tag_V2" : Int = PLC Recipe_db.Velocity_array[1] AT %MW68, 1 s
   "HMI_Tag_V3" : Int = PLC Recipe_db.Velocity_array[2] AT %MW72, 1 s
   "HMI_Tag_V4" : Int = PLC Recipe_db.Velocity_array[3] AT %MW76, 1 s
   "HMI_Tag_V5" : Int = PLC Recipe_db.Velocity_array[4] AT %MW80, 1 s
   "HMI_Tag_V6" : Int = PLC Recipe_db.Velocity_array[5] AT %MW84, 1 s
   "RecipeNumber" : Int AT %DB1.DBW0
   "HMI_Tag_T7" : Int = PLC Recipe_db.Time_array[6] AT %DB1.DBW0, 1 s
   "HMI_Tag_T8" : Int = PLC Recipe_db.Time_array[7] AT %DB1.DBW0, 1 s
   "HMI_Tag_T9" : Int = PLC Recipe_db.Time_array[8] AT %DB1.DBW0, 1 s
   "HMI_Tag_T10" : Int = PLC Recipe_db.Time_array[9] AT %DB1.DBW0, 1 s
   "HMI_Tag_T11" : Int = PLC Recipe_db.Time_array[10] AT %DB1.DBW0, 1 s
   "HMI_Tag_T12" : Int = PLC Recipe_db.Time_array[11] AT %DB1.DBW0, 1 s
   "HMI_Tag_T13" : Int = PLC Recipe_db.Time_array[12] AT %DB1.DBW0, 1 s
   "HMI_Tag_V7" : Int = PLC Recipe_db.Velocity_array[6] AT %DB1.DBW0, 1 s
   "HMI_Tag_V8" : Int = PLC Recipe_db.Velocity_array[7] AT %DB1.DBW0, 1 s
   "HMI_Tag_V9" : Int = PLC Recipe_db.Velocity_array[8] AT %DB1.DBW0, 1 s
   "HMI_Tag_V10" : Int = PLC Recipe_db.Velocity_array[9] AT %DB1.DBW0, 1 s
   "HMI_Tag_V11" : Int = PLC Recipe_db.Velocity_array[10] AT %DB1.DBW0, 1 s
   "HMI_Tag_V12" : Int = PLC Recipe_db.Velocity_array[11] AT %DB1.DBW0, 1 s
   "HMI_Tag_V13" : Int = PLC Recipe_db.Velocity_array[12] AT %DB1.DBW0, 1 s

recipe "Recipe_1": Recipe_element_1 <- "HMI_Tag_T1", Recipe_element_2 <- "HMI_Tag_V1", Recipe_element_3 <- "HMI_Tag_T2", Recipe_element_4 <- "HMI_Tag_V2", Recipe_element_5 <- "HMI_Tag_T3", Recipe_element_6 <- "HMI_Tag_V3", Recipe_element_7 <- "HMI_Tag_T4", Recipe_element_8 <- "HMI_Tag_V4", Recipe_element_9 <- "HMI_Tag_T5", Recipe_element_10 <- "HMI_Tag_V5", Recipe_element_11 <- "HMI_Tag_T6", Recipe_element_12 <- "HMI_Tag_V6"

Template "Template_1" 1280x740
   Button "Start screen" at 1200,3 size 78x59; TextOff 'Start screen'; PictureOff "NavigateHome_TP1200_Comfort_TR"; PictureOn "NavigateHome_TP1200_Comfort_TR"
      on Release: ActivateScreen("Root screen", 0)
   Button "Template_Button" at 1200,64 size 78x59; TextOff 'Tryb ręczny'; PictureOff "Navigates to System information for TP1200 Comfort 17.0.0.0"
      on Click: ActivateScreen("manual_mode", 0)
   Button "Template_Button_1" at 1200,126 size 78x59; TextOff 'Tryb auto.'
      on Click: ActivateScreen("automatic_mode", 0)
   Button "Template_Button_3" at 1200,249 size 78x59; TextOff 'Text'
   Button "Template_Button_4" at 1200,310 size 78x59; TextOff 'Text'
   Button "Template_Button_5" at 1200,372 size 78x59; TextOff 'Text'
   Button "Exit" at 1200,679 size 78x59; TextOff 'Exit'; PictureOff "ExitRuntime_TP1200_Comfort_TR"; PictureOn "ExitRuntime_TP1200_Comfort_TR"
      on Release: StopRuntime(0)
   Button "Log on" at 1200,618 size 78x59; TextOff 'Log on'; PictureOff "Login_TP1200_Comfort_TR"; PictureOn "Login_TP1200_Comfort_TR"
      on Release: function_a2a04561(); function_f41c6f6c("HMI_Tag_temp_login"); function_e1ab61de("HMI_Tag_1_temp_user_number")
   AlarmView "Alarm view_Unacknowledged" at 0,0 size 1201x23
   Button "Template_Button_8" at 1200,188 size 78x59; TextOff 'Text'; PictureOff "Graphic_3"
      on Click: ActivateScreen("recipes", 0)
   Button "Template_Button_9" at 1200,433 size 78x59; TextOff 'Text'
      on Click: ActivateScreen("Alarms", 0)
   Button "Template_Button_10" at 1200,494 size 78x59; TextOff 'Text'
   Button "Language_1" at 1199,556 size 78x59; TextOn 'Language'; TextOff 'Text'; PictureOn "ToggleLanguage_TP1200_Comfort_TR"; PictureOff "Graphic_4"
      on Release: function_fb9197e8(-1)
   Button "Template_Button_2" at 1200,188 size 78x59; TextOff 'Text'
      on Click: ActivateScreen("recipes", 0)
      ObjectEnable <- "HMI_Tag_1_temp_user_number"
   Button "Template_Button_6" at 1200,433 size 78x59; TextOff 'Text'
      on Click: ActivateScreen("Alarms", 0)
   Button "Template_Button_7" at 1200,494 size 78x59; TextOff 'Text'
      on Click: ActivateScreen("User administration", 0)
   Button "Language" at 1200,557 size 78x59; TextOff 'Text'; TextOn 'Language'; PictureOn "ToggleLanguage_TP1200_Comfort_TR"; PictureOff "Graphic_4"
      on Click: ActivateScreen("System settings", 0)
   GraphicView "Template_Graphic view_3" at 1213,439 size 56x47; Picture "Graphic_5"
   GraphicView "Template_Graphic view_4" at 1200,503 size 59x42; Picture "Graphic_6"
   GraphicView "Template_Graphic view_2" at 1215,563 size 49x47; Picture "Graphic_4"
   GraphicView "Template_Graphic view_1" at 1216,197 size 47x42; Picture "Graphic_3"
      Visibility <- "HMI_Tag_1_temp_user_number"
   GraphicView "Template_Graphic view_5" at 1237,519 size 36x30; Picture "Graphic_7"

screen "Root screen" 1280x740, template "Template_1"
   on GenerateScreen: SetTag("Tag_ScreenNumber", 1)
   Button "Button_1" at 970,35 size 218x75; TextOff 'Logowanie'
      on Release: function_a2a04561(); function_f41c6f6c("HMI_Tag_temp_login"); function_e1ab61de("HMI_Tag_1_temp_user_number")
      Visibility <- "HMI_Tag_1_temp_user_number"
   TextField "Text field_1" at 134,161 size 517x28; Text 'Stanowisko do testów przekładni kolejowych.'
   TextField "Text field_2" at 136,200 size 927x25; Text 'W celu wykonania testów według predefiniowanych nastaw prosze wybrać "Tryb automatyczny".'
   TextField "Text field_3" at 132,266 size 1022x46; Text 'W celu edycji predefiniowanych nastaw należy być zalogowanym na konto z odpowiednimi uprawnieniami a nastepnie wybrać przycisk "Zarządzanie parametrami".'
   Button "Button_2" at 105,519 size 306x89; TextOff 'Tryb automatyczny'
      on Click: ActivateScreen("automatic_mode", 0)
   Button "Button_4" at 438,519 size 306x89; TextOff 'Tryb ręczny'
      on Click: ActivateScreen("manual_mode", 0)
   Button "Button_5" at 785,519 size 306x89; TextOff 'Zarządzanie recepturami'
      Visibility <- "HMI_Tag_1_temp_user_number"
      on Click: ActivateScreen("recipes", 0)
   Button "Button_3" at 970,35 size 218x75; TextOff 'Wyloguj'
      on Release: function_f23ef4c9(); function_f41c6f6c("HMI_Tag_temp_login"); function_e1ab61de("HMI_Tag_1_temp_user_number")
      Visibility <- "HMI_Tag_1_temp_user_number"

screen "System screens" 1280x740, template "Template_1"
   on GenerateScreen: SetTag("Tag_ScreenNumber", 2)
   Button "Back" at 1,25 size 159x47; TextOff 'Back'
      on Release: ActivateScreen("Root screen", 0)
   Button "HmiScreenItemData" at 36,119 size 159x47; TextOff 'SIMATIC PLC system diagnos...'; PictureOff "Navigates to SIMATIC PLC system diagnostics for TP1200 Comfort 17.0.0.0"; PictureOn "Navigates to SIMATIC PLC system diagnostics for TP1200 Comfort 17.0.0.0"
      on Release: ActivateScreen("SIMATIC PLC system diagnostics", 0)
   Button "HmiScreenItemData_1" at 36,178 size 159x47; TextOff 'Project information'; PictureOff "Navigates to Project information for TP1200 Comfort 17.0.0.0"; PictureOn "Navigates to Project information for TP1200 Comfort 17.0.0.0"
   Button "HmiScreenItemData_2" at 36,237 size 159x47; TextOff 'System settings'; PictureOff "Navigates to System settings for TP1200 Comfort 17.0.0.0"; PictureOn "Navigates to System settings for TP1200 Comfort 17.0.0.0"
      on Release: ActivateScreen("System settings", 0)
   Button "HmiScreenItemData_3" at 36,296 size 159x47; TextOff 'User administration'; PictureOff "Navigates to User administration for TP1200 Comfort 17.0.0.0"; PictureOn "Navigates to User administration for TP1200 Comfort 17.0.0.0"
      on Release: ActivateScreen("User administration", 0)
   Button "HmiScreenItemData_4" at 36,355 size 159x47; TextOff 'System information'; PictureOff "Navigates to System information for TP1200 Comfort 17.0.0.0"; PictureOn "Navigates to System information for TP1200 Comfort 17.0.0.0"
   Button "HmiScreenItemData_5" at 36,414 size 159x47; TextOff 'Different jobs'; PictureOff "Navigates to Different jobs for TP1200 Comfort 17.0.0.0"; PictureOn "Navigates to Different jobs for TP1200 Comfort 17.0.0.0"
      on Release: ActivateScreen("Different jobs", 0)

screen "SIMATIC PLC system diagnostics" 1280x740, template "Template_1"
   on GenerateScreen: SetTag("Tag_ScreenNumber", 3)
   SysDiagControl "HmiScreenItemData" at 1,73 size 1197x659
   Button "Back" at 1,25 size 159x47; TextOff 'Back'
      on Release: ActivateScreen("System screens", 0)

